BC00170=183095,975695,1075175
BC00171=183095,975695,1075175
BC00172=183095,975695,1075175
BC00173=183095,975695,1075175
BC00174=183095,975695,1075175
BC00175=183095,975695,1075175
BC00176=183095,975695,1075175
BC00177=183095,975695,1075175
BC00178=183095,975695,1075175
BC00179=210625,968928,1075175
BC00180=210625,968928,1075175
BC00181=210625,968928,1075175
BC00182=210625,968928,1075175
BC00183=210625,968928,1075175
BC00184=210625,968928,1075175
BC00185=210625,968928,1075175
BC00186=180246,951709,1075175
BC00187=180247,951710,1075174
BC00188=180247,951710,1075174
BC00189=180247,951710,1075174
BC00190=180247,951710,1075174
BC00191=180247,951710,1075174
BC00192=180247,951710,1075174
BC00193=180247,951710,1075174
BC00194=180247,951710,1075174
BC00195=180247,951710,1075174
BC00196=220770,956468,1075173
BC00197=254413,953027,1075175
BC00198=252547,954523,1075175
BC00199=252548,954519,1075175
BC00200=252583,954651,1075175
BC00201=252019,957675,1075175
BC00202=252583,954651,1075175
BC00203=252165,954787,1075175
BC00204=249030,954243,1075175
BC00205=252165,954787,1075175
BC00206=258696,949550,1075175
BC00207=257059,950024,1075175
BC00208=265795,953000,1075175
BC00209=262609,959912,1075175
BC00210=262609,959912,1075175
BC00211=262609,959912,1075175
BC00212=262609,959912,1075175
BC00213=262609,959912,1075175
BC00214=219729,982607,1075175
BC00215=219729,982607,1075175
BC00216=219729,982607,1075175
BC00217=219729,982607,1075175
BC00218=219729,982607,1075175
BC00219=219729,982607,1075175
BC00220=219729,982607,1075175
BC00221=219729,982607,1075175
BC00222=219729,982607,1075175
BC00223=219729,982607,1075175
BC00224=247259,975840,1075175
BC00225=247259,975840,1075175
BC00226=247259,975840,1075175
BC00227=247259,975840,1075175
BC00228=247259,975840,1075175
BC00229=247259,975840,1075175
BC00230=247259,975840,1075175
BC00231=216880,958621,1075175
BC00232=216881,958622,1075174
BC00233=216881,958622,1075174
BC00234=216881,958622,1075174
BC00235=216881,958622,1075174
BC00236=216881,958622,1075174
BC00237=216881,958622,1075174
BC00238=216881,958622,1075174
BC00239=216881,958622,1075174
BC00240=216881,958622,1075174
BC00241=254634,951648,1075175
BC00242=254634,951649,1075174
BC00243=254634,951649,1075174
BC00244=207516,961105,1075174
BC00245=207516,961105,1075174
BC00246=207516,961105,1075174
BC00247=207516,961105,1075174
BC00248=207516,961105,1075174
BC00249=207516,961105,1075174
BC00250=207516,961105,1075174
BC00251=207516,961105,1075174
BC00252=207675,961073,1075174
BC00253=248439,993035,1075175
BC00254=271638,1017285,1075175
BC00255=314947,1062557,1075175
BC00256=311280,1056373,1075175
BC00257=310409,1054905,1075175
BC00258=310409,1054901,1075175
BC00259=310409,1054905,1075175
BC00260=284329,1066137,1075175
BC00261=285931,1063482,1075175
BC00262=284329,1066137,1075175
BC00263=333588,1039325,1075175
BC00264=330835,1037779,1075175
BC00265=333588,1039325,1075175
BC00266=340460,1045393,1075175
BC00267=319968,1046454,1075175
BC00268=297161,1046455,1075174
BC00269=305514,1060044,1075174
BC00270=305514,1060044,1075174
BC00271=305514,1060044,1075174
BC00272=305514,1060044,1075174
BC00273=270133,1060044,1075174
BC00274=270133,1060044,1075174
BC00275=270133,1060044,1075174
BC00276=270133,1060044,1075174
BC00277=270133,1060044,1075174
BC00278=271678,1058058,1075174
BC00279=253507,1028204,1074244
BC00280=253507,1028204,1074244
BC00281=253507,1028204,1074244
BC00282=253507,1028204,1074244
BC00283=253507,1028204,1074244
BC00284=253507,1028204,1074244
BC00285=253507,1028204,1074244
BC00286=253507,1028204,1074244
BC00287=253507,1028204,1074244
BC00288=253507,1028204,1074244
BC00289=253507,1028204,1074244
BC00290=253507,1028204,1074244
BC00291=253507,1028204,1074244
BC00292=212842,1022781,1075175
BC00293=146334,1015862,1075175
BC00294=66205,1045023,1075175
BC00295=66205,1045023,1075175
BC00296=66205,1045023,1075175
BC00297=66205,1045023,1075175
BC00298=66205,1045023,1075175
BC00299=66205,1045023,1075175
BC00300=66205,1045023,1075175
BC00301=66205,1045023,1075175
BC00302=66205,1045023,1075175
BC00303=66205,1045023,1075175
BC00304=66205,1045023,1075175
BC00305=66205,1045023,1075175
BC00306=125029,959783,1075175
BC00307=190390,972133,1075175
BC00308=190390,972133,1075175
BC00309=190390,972133,1075173
BC00310=190390,972133,1075175
BC00311=190390,972133,1075175
BC00312=190390,972133,1075175
BC00313=190390,972133,1075175
BC00314=190390,972133,1075175
BC00315=190390,972133,1075175
BC00316=190390,972133,1075175
BC00317=190390,972133,1075175
BC00318=190390,972133,1075175
BC00319=190390,972133,1075175
BC00320=163122,952799,1075175
BC00321=172813,952714,1075175
BC00322=172813,952714,1075175
BC00323=172813,952714,1075175
BC00324=172813,952714,1075175
BC00325=172813,952714,1075175
BC00326=172813,952714,1075175
BC00327=172813,952714,1075175
BC00328=172813,952714,1075175
BC00329=172813,952714,1075175
BC00330=172813,952714,1075175
BC00331=172813,952714,1075175
BC00332=172813,952714,1075175
BC00333=172813,952714,1075175
BC00334=167655,947910,1075175
BC00335=103363,888035,1075175
BC00336=35304,822265,1075175
BC00337=60536,839097,1075175
BC00338=60536,839097,1075175
BC00339=60536,839097,1075175
BC00340=60536,839097,1075175
BC00341=60536,839097,1075175
BC00342=60536,839097,1075175
BC00343=35912,824089,1075175
BC00344=35912,824089,1075175
BC00345=35912,824089,1075175
BC00346=35912,824089,1075175
BC00347=35912,824089,1075175
BC00348=35912,824089,1075175
BC00349=35304,822265,1075175
BC00350=35304,822265,1075175
BC00351=35304,822265,1075175
BC00352=35304,822265,1075175
BC00353=35304,822265,1075175
BC00354=35304,822265,1075175
BC00355=35304,822265,1075175
BC00356=35304,822265,1075175
BC00357=35304,822265,1075175
BC00358=35304,822265,1075175
BC00359=35304,822265,1075175
BC00360=167967,799945,1075175
BC00361=311305,898961,1075175
BC00362=311305,898961,1075175
BC00363=311305,898961,1075175
BC00364=311305,898961,1075175
BC00365=311305,898961,1075175
BC00366=311305,898961,1075175
BC00367=311305,898961,1075175
BC00368=311305,898961,1075175
BC00369=311305,898961,1075175
BC00370=311305,898961,1075175
BC00371=311305,898961,1075175
BC00372=311305,898961,1075175
BC00373=113180,824290,1075229
BC00374=113180,824290,1075229
BC00375=113180,824290,1075229
BC00376=113180,824290,1075229
BC00377=113180,824290,1075229
BC00378=113180,824290,1075229
BC00379=113180,824290,1075229
BC00380=113180,824290,1075229
BC00381=113180,824290,1075229
BC00382=113180,824290,1075229
BC00383=113180,824290,1075229
BC00384=113180,824290,1075229
BC00385=355762,967535,1075175
BC00386=355762,967535,1075175
BC00387=355762,967535,1075175
BC00388=355762,967535,1075175
BC00389=355762,967535,1075175
BC00390=355762,967535,1075175
BC00391=355762,967535,1075175
BC00392=355762,967535,1075175
BC00393=397203,974799,1075175
BC00394=397203,974799,1075175
BC00395=397203,974799,1075175
BC00396=397203,974799,1075175
BC00397=397203,974799,1075175
BC00398=397203,974799,1075175
BC00399=397203,974799,1075175
BC00400=397203,974799,1075175
BC00401=389868,1004990,1075175
BC00402=389868,1004990,1075175
BC00403=389868,1004990,1075175
BC00404=389868,1004990,1075175
BC00405=389868,1004990,1075175
BC00406=389868,1004990,1075175
BC00407=397203,974799,1075175
BC00408=279782,952911,1075175
BC00409=264332,967435,1075175
BC00410=264332,967435,1075175
BC00411=264332,967435,1075175
BC00412=264332,967435,1075175
BC00413=264332,967435,1075175
BC00414=264332,967435,1075175
BC00415=264332,967435,1075175
BC00416=264332,967435,1075175
BC00417=264332,967435,1075175
BC00418=264332,967435,1075175
BC00419=264332,967435,1075175
BC00420=290594,956201,1075175
BC00421=316856,944967,1075175
BC00422=316856,944967,1075175
BC00423=316856,944967,1075175
BC00424=316856,944967,1075175
BC00425=316856,944967,1075175
BC00426=316856,944967,1075175
BC00427=316856,944967,1075175
BC00428=316856,944967,1075175
BC00429=316856,944967,1075175
BC00430=316856,944967,1075175
BC00431=316856,944967,1075175
BC00432=316856,944967,1075175
BC00433=316856,944967,1075175
BC00434=316856,944967,1075175
BC00435=316856,944967,1075175
BC00436=316856,944967,1075175
BC00437=329946,891084,1075175
BC00438=337525,859888,1075175
BC00439=337525,859888,1075175
BC00440=337525,859888,1075175
BC00441=337525,859888,1075175
BC00442=337525,859888,1075175
BC00443=337525,859888,1075175
BC00444=337525,859888,1075175
BC00445=337525,859888,1075175
BC00446=238148,874377,1075175
BC00447=227206,875826,1075175
BC00448=227206,875826,1075175
BC00449=227206,875826,1075175
BC00450=227206,875826,1075175
BC00451=227206,875826,1075175
BC00452=227206,875826,1075175
BC00453=280946,887675,1075175
BC00454=280946,887675,1075175
BC00455=280946,887675,1075175
BC00456=280946,887675,1075175
BC00457=280946,887675,1075175
BC00458=280946,887675,1075175
BC00459=280946,887675,1075175
BC00460=280946,887675,1075175
BC00461=239261,850045,1075175
BC00462=207869,857354,1075175
BC00463=207869,857354,1075175
BC00464=207869,857354,1075175
BC00465=207869,857354,1075175
BC00466=207869,857354,1075175
BC00467=207869,857354,1075175
BC00468=207869,857354,1075175
BC00469=207869,857354,1075175
BC00470=207996,857850,1075175
BC00471=184532,936508,1075175
BC00472=203495,1021788,1075175
BC00473=203934,1024782,1075175
BC00474=204108,1022909,1075171
BC00475=204109,1022908,1075172
BC00476=193998,1019034,1075175
BC00477=193559,1023720,1075175
BC00478=122539,997675,1075175
BC00479=122539,997675,1075175
BC00480=122540,997675,1075169
BC00481=122540,997675,1075169
BC00482=122539,997675,1075175
BC00483=122539,997675,1075175
BC00484=110261,971952,1075175
BC00485=110261,971952,1075175
BC00486=110261,971952,1075175
BC00487=110261,971952,1075175
BC00488=110261,971952,1075175
BC00489=110261,971952,1075175
BC00490=222038,980891,1075175
BC00491=314817,1023461,1075175
BC00492=333143,1031869,1075175
BC00493=333143,1031869,1075175
BC00494=333143,1031869,1075175
BC00495=333143,1031869,1075175
BC00496=333143,1031869,1075175
BC00497=163675,1006427,1075175
BC00498=163675,1006427,1075175
BC00499=164114,1001741,1075175
BC00500=164289,999867,1075175
BC00501=160191,997498,1075175
BC00502=158450,996490,1075175
BC00503=154353,994119,1075175
BC00504=154178,995993,1075175
BC00505=153739,1000679,1075175
BC00506=82719,974634,1075175
BC00507=82719,974634,1075175
BC00508=82720,974634,1075172
BC00509=82720,974634,1075172
BC00510=82719,974634,1075175
BC00511=82720,974634,1075173
BC00512=82719,974634,1075175
BC00513=82719,974634,1075175
BC00514=70441,948911,1075175
BC00515=70441,948911,1075175
BC00516=70441,948911,1075175
BC00517=70441,948911,1075175
BC00518=70441,948911,1075175
BC00519=70441,948911,1075175
BC00520=182218,957850,1075175
BC00521=274997,1000420,1075175
BC00522=293323,1008828,1075175
BC00523=293323,1008828,1075175
BC00524=293323,1008828,1075175
BC00525=293323,1008828,1075175
BC00526=293323,1008828,1075175
BC00527=293323,1008828,1075175
BC00528=337244,1059629,1075175
BC00529=337244,1059629,1075175
BC00530=337244,1059629,1075175
BC00531=337244,1059629,1075175
BC00532=337244,1059629,1075175
BC00533=337244,1059629,1075175
BC00534=337244,1059629,1075175
BC00535=227430,982125,1075175
BC00536=115014,939685,1075175
BC00537=118867,937244,1075175
BC00538=120408,936268,1075175
BC00539=124434,938528,1075175
BC00540=125926,939366,1075175
BC00541=125926,939366,1075175
BC00542=140995,947826,1075175
BC00543=140995,947826,1075175
BC00544=182041,976368,1075174
BC00545=182041,976368,1075174
BC00546=180846,977671,1075175
BC00547=177859,980929,1075175
BC00548=194800,984537,1075175
BC00549=244653,1016084,1075175
BC00550=241511,1010564,1075175
BC00551=240254,1008357,1075175
BC00552=240254,1008354,1075175
BC00553=241511,1010562,1075175
BC00554=244653,1016081,1075175
BC00555=244653,1016084,1075175
BC00556=272695,1033702,1075175
BC00557=285514,1041756,1075175
BC00558=284751,1045931,1075175
BC00559=282162,1039999,1075175
BC00560=281126,1037626,1075175
BC00561=207140,1028015,1075175
BC00562=213441,1031536,1075175
BC00563=213388,1030834,1075175
BC00564=213388,1030834,1075175
BC00565=212628,1031081,1075217
BC00566=212628,1031081,1075217
BC00567=212628,1031081,1075217
BC00568=212628,1031081,1075217
BC00569=212628,1031081,1075202
BC00570=202210,1012854,1075175
BC00571=202210,1012854,1075175
BC00572=208776,1017549,1075175
BC00573=200305,979606,1075175
BC00574=185662,909371,1075175
BC00575=185662,823633,1075175
BC00576=152631,778532,1075175
BC00577=146092,780306,1075175
BC00578=143477,781016,1075175
BC00579=143597,781078,1075175
BC00580=143625,781092,1075175
BC00581=143746,781156,1075175
BC00582=146361,780446,1075175
BC00583=152900,778672,1075175
BC00584=152900,778672,1075175
BC00585=74084,744686,1075175
BC00586=74084,744686,1075175
BC00587=67287,679894,1075175
BC00588=67287,679894,1075175
BC00589=67287,679894,1075175
BC00590=67287,679894,1075175
BC00591=67287,679894,1075175
BC00592=67287,679894,1075175
BC00593=67287,679894,1075175
BC00594=67287,679894,1075175
BC00595=83395,694294,1075175
BC00596=102108,711022,1075175
BC00597=165558,767742,1075175
BC00598=222482,818628,1075175
BC00599=215814,820321,1075175
BC00600=213147,820999,1075175
BC00601=213147,820994,1075175
BC00602=213147,820993,1075175
BC00603=213148,820988,1075175
BC00604=215815,820311,1075175
BC00605=222483,818617,1075175
BC00606=173722,816110,1075175
BC00607=90356,811823,1075175
BC00608=89696,811574,1075175
BC00609=89432,811475,1075175
BC00610=89432,811475,1075175
BC00611=89432,811475,1075175
BC00612=85301,809160,1075175
BC00613=73323,802435,1075175
BC00614=69196,800114,1075175
BC00615=69460,800213,1075175
BC00616=70120,800462,1075175
BC00617=203969,867991,1075175
BC00618=200192,866637,1075175
BC00619=198681,866095,1075175
BC00620=196278,870078,1075175
BC00621=188025,883752,1075175
BC00622=185620,887734,1075175
BC00623=187131,888276,1075175
BC00624=190907,889630,1075175
BC00625=185807,834457,1075175
BC00626=185042,826181,1075175
BC00627=182820,831186,1075175
BC00628=181931,833188,1075174
BC00629=181931,833188,1075174
BC00630=205283,846231,1075175
BC00631=205283,846231,1075175
BC00632=246906,863634,1075175
BC00633=246906,863634,1075175
BC00634=248214,861732,1075175
BC00635=251484,856977,1075175
BC00636=177002,833071,1075175
BC00637=153563,828435,1075175
BC00638=140020,825224,1075175
BC00639=143607,831260,1075175
BC00640=145042,833675,1075175
BC00641=145042,833675,1075175
BC00642=143607,831255,1075175
BC00643=140021,825218,1075175
BC00644=140020,825224,1075175
BC00645=325300,955877,1075175
BC00646=326098,960603,1075175
BC00647=326417,962494,1075175
BC00648=373942,970744,1075175
BC00649=373934,970699,1075175
BC00650=373927,970659,1075175
BC00651=372825,964128,1075175
BC00652=388713,844195,1075175
BC00653=388713,844195,1075175
BC00654=388713,844195,1075175
BC00655=388713,844195,1075175
BC00656=388713,844195,1075175
BC00657=392621,845560,1075175
BC00658=388844,869736,1075175
BC00659=388844,869736,1075175
BC00660=388844,869736,1075175
BC00661=388844,869736,1075175
BC00662=386515,859937,1075175
BC00663=382579,861240,1075175
BC00664=382579,861240,1075175
BC00665=398174,862085,1075175
BC00666=398174,860729,1075175
BC00667=398175,860364,1075172
BC00668=398174,860364,1075175
BC00669=398174,860364,1075175
BC00670=398174,860364,1075175
BC00671=398174,859798,1075175
BC00672=398174,853900,1075175
BC00673=335556,962122,1075175
BC00674=313093,960913,1075175
BC00675=312779,966350,1075175
BC00676=312653,968525,1075175
BC00677=312653,968525,1075175
BC00678=313384,968652,1075175
BC00679=313384,968652,1075175
BC00680=322722,968076,1075175
BC00681=323035,962639,1075175
BC00682=275790,965253,1075175
BC00683=219096,968390,1075175
BC00684=223120,970377,1075175
BC00685=224729,971172,1075175
BC00686=224729,971172,1075175
BC00687=224591,971007,1075175
BC00688=224591,971007,1075175
BC00689=219210,965708,1075175
BC00690=215186,963721,1075175
BC00691=283252,975030,1075175
BC00692=343583,985054,1075175
BC00693=351318,986339,1075175
BC00694=346951,987672,1075175
BC00695=346840,986833,1075175
BC00696=346840,986833,1075175
BC00697=346840,986832,1075174
BC00698=346840,986832,1075174
BC00699=346840,986832,1075174
BC00700=351469,983882,1075175
BC00701=355836,982549,1075175
BC00702=351318,986339,1075175
BC00703=375376,962122,1075175
BC00704=352913,960913,1075175
BC00705=352599,966350,1075175
BC00706=352473,968525,1075175
BC00707=352473,968525,1075175
BC00708=352749,968573,1075175
BC00709=352749,968573,1075175
BC00710=362542,968076,1075175
BC00711=362855,962639,1075175
BC00712=315610,965253,1075175
BC00713=258916,968390,1075175
BC00714=262940,970377,1075175
BC00715=264549,993234,1075175
BC00716=264533,993126,1075175
BC00717=264533,993126,1075175
BC00718=264533,993126,1075175
BC00719=259030,965708,1075175
BC00720=255006,963721,1075175
BC00721=323072,975030,1075175
BC00722=383403,985054,1075175
BC00723=391138,986339,1075175
BC00724=386771,987672,1075175
BC00725=385397,987893,1075175
BC00726=385397,987893,1075175
BC00727=385397,987893,1075175
BC00728=385397,987893,1075175
BC00729=391289,983882,1075175
BC00730=394785,983280,1075175
BC00731=393350,984484,1075175
BC00732=322594,894090,1075175
BC00733=319270,885244,1075175
BC00734=319145,881395,1075175
BC00735=319096,879856,1075175
BC00736=319096,879856,1075175
BC00737=310158,881364,1075175
BC00738=310282,885213,1075175
BC00739=287932,898047,1075175
BC00740=289217,893542,1075175
BC00741=289730,891739,1075175
BC00742=285692,891718,1075175
BC00743=285179,893520,1075175
BC00744=283894,898026,1075175
BC00745=317886,904348,1075175
BC00746=321408,904356,1075175
BC00747=251917,914686,1075175
BC00748=191223,885215,1075175
BC00749=191223,923708,1075175
BC00750=186619,926680,1075175
BC00751=184777,927869,1075175
BC00752=132357,904545,1075175
BC00753=148459,907340,1075175
BC00754=150318,907039,1075175
BC00755=172119,903510,1075175
BC00756=172334,901853,1075175
BC00757=172871,897709,1075175
BC00758=285135,920733,1075175
BC00759=282294,924718,1075175
BC00760=278369,925274,1075175
BC00761=250842,915028,1075175
BC00762=259644,916574,1075175
BC00763=259644,916574,1075174
BC00764=259644,916574,1075175
BC00765=285135,920733,1075175
BC00766=320470,920733,1075175
BC00767=320470,920733,1075175
BC00768=320470,920733,1075172
BC00769=320470,920733,1075172
BC00770=320470,920733,1075172
BC00771=302481,924098,1075175
BC00772=235391,926007,1075175
BC00773=235391,926007,1075175
BC00774=227742,920504,1075175
BC00775=172871,874776,1075175
BC00776=140749,823212,1075175
BC00777=114392,780903,1075175
BC00778=114392,780903,1075175
BC00779=114392,780903,1075175
BC00780=114392,780903,1075175
BC00781=114393,780903,1075175
BC00782=114392,780903,1075175
BC00783=114392,780903,1075175
BC00784=114392,780903,1075175
BC00785=147421,791636,1075175
BC00786=157474,794903,1075175
BC00787=157474,794903,1075175
BC00788=157474,794903,1075174
BC00789=157474,794903,1075175
BC00790=157474,794903,1075175
BC00791=157474,794903,1075175
BC00792=157474,794903,1075175
BC00793=157474,794903,1075175
BC00794=188976,808930,1075175
BC00795=188976,808930,1075175
BC00796=188976,808930,1075175
BC00797=188976,808930,1075175
BC00798=188976,808930,1075175
BC00799=188976,808930,1075175
BC00800=188976,808930,1075175
BC00801=188976,808930,1075175
BC00802=147641,782026,1075175
BC00803=198576,845167,1075175
BC00804=232811,933878,1075175
BC00805=232896,933343,1075175
BC00806=232035,938717,1075175
BC00807=231691,940867,1075175
BC00808=233684,941999,1075172
BC00809=218918,951560,1075175
BC00810=218487,945823,1075175
BC00811=199715,965567,1075175
BC00812=202231,971242,1075175
BC00813=203237,973512,1075175
BC00814=199770,971953,1075175
BC00815=198686,969649,1075175
BC00816=195975,963887,1075175
BC00817=268319,958805,1075175
BC00818=299772,956595,1075175
BC00819=294961,960779,1075175
BC00820=302025,967105,1075175
BC00821=302025,967105,1075175
BC00822=302862,967571,1075175
BC00823=304981,965989,1075175
BC00824=310277,962032,1075175
BC00825=299772,946803,1075175
BC00826=156368,867370,1075175
BC00827=114190,943890,1075175
BC00828=112857,947238,1075175
BC00829=112324,948578,1075175
BC00830=112324,948578,1075175
BC00831=97258,945962,1075175
BC00832=58795,939285,1075175
BC00833=58795,939285,1075175
BC00834=57972,937710,1075175
BC00835=59304,934362,1075175
BC00836=59959,931573,1075175
BC00837=60163,930702,1075175
BC00838=64900,934429,1075175
BC00839=66794,935919,1075175
BC00840=70926,933782,1075175
BC00841=86714,920781,1075175
BC00842=88876,916896,1075175
BC00843=87247,915034,1075175
BC00844=83174,910378,1075175
BC00845=93083,910762,1075175
BC00846=96362,916987,1075175
BC00847=99439,917931,1075175
BC00848=102107,915596,1075175
BC00849=93734,925368,1075175
BC00850=92128,923198,1075175
BC00851=88115,917772,1075175
BC00852=59304,853852,1075175
BC00853=302197,956351,1075175
BC00854=302197,956351,1075175
BC00855=297684,958955,1075175
BC00856=295879,959997,1075175
BC00857=304739,998959,1075175
BC00858=304739,998896,1075175
BC00859=293949,1042099,1075175
BC00860=295296,1044279,1075175
BC00861=298665,1049727,1075175
BC00862=298665,1049727,1075175
BC00863=302197,956351,1075175
BC00864=339931,956351,1075175
BC00865=339931,956351,1075175
BC00866=339931,956351,1075175
BC00867=345108,996833,1075175
BC00868=329498,1037164,1075167
BC00869=329498,1037164,1075167
BC00870=329498,1037164,1075167
BC00871=326051,1024211,1075168
BC00872=315665,949153,1075168
BC00873=252444,896504,1075168
BC00874=116643,896504,1075168
BC00875=116643,972299,1075168
BC00876=116644,972299,1070754
BC00877=116644,972299,1070754
BC00878=121804,1001122,1070754
BC00879=121804,1001122,1070754
BC00880=121804,1001122,1070754
BC00881=121804,1001122,1070754
BC00882=164206,909682,1070754
BC00883=118737,834368,1072160
BC00884=21214,672831,1075175
BC00885=78393,670967,1075175
BC00886=177059,727519,1002542
BC00887=78393,913126,1075175
BC00888=70793,903989,1075175
BC00889=70793,903989,1075175
BC00890=70793,903989,1075175
BC00891=70793,903989,1075175
BC00892=70793,903989,1075175
BC00893=70793,903989,1075175
BC00894=70793,903989,1075175
BC00895=70793,903989,1075175
BC00896=70793,903989,1075175
BC00897=103901,897249,1075175
BC00898=103901,897249,1075175
BC00899=103901,897249,1075175
BC00900=103901,897249,1075175
BC00901=103901,897249,1075175
BC00902=103901,897249,1075175
BC00903=103901,897249,1075175
BC00904=103901,897249,1075175
BC00905=89915,910531,1075175
BC00906=89915,910531,1075175
BC00907=89915,910531,1075175
BC00908=89915,910531,1075175
BC00909=89915,910531,1075175
BC00910=89915,910531,1075175
BC00911=89915,910531,1075175
BC00912=89915,910531,1075175
BC00913=89915,910531,1075175
BC00914=27368,899646,1075175
BC00915=27368,899646,1075175
BC00916=27368,899646,1075175
BC00917=27368,899646,1075175
BC00918=27368,899646,1075175
BC00919=27368,899646,1075175
BC00920=27368,899646,1075175
BC00921=27368,899646,1075175
BC00922=160753,772187,1075175
BC00923=160753,772187,1075175
BC00924=160753,772187,1075175
BC00925=160753,772187,1075175
BC00926=160753,772187,1075175
BC00927=160753,772187,1075175
BC00928=160753,772187,1075175
BC00929=160753,772187,1075175
BC00930=160753,772187,1075175
BC00931=160753,772187,1075175
BC00932=160753,772187,1075175
BC00933=160753,772187,1075175
BC00934=123402,765716,1075175
BC00935=123402,765716,1075175
BC00936=123402,765716,1075175
BC00937=123402,765716,1075175
BC00938=123402,765716,1075175
BC00939=123402,765716,1075175
BC00940=123402,765716,1075175
BC00941=123402,765716,1075175
BC00942=123402,765716,1075175
BC00943=123402,765716,1075175
BC00944=123402,765716,1075175
BC00945=129464,768278,1075175
BC00946=151149,777443,1075175
BC00947=169689,785624,1075175
BC00948=169689,785624,1075175
BC00949=169689,785624,1075175
BC00950=169689,785624,1075175
BC00951=169689,785624,1075175
BC00952=169689,785624,1075175
BC00953=169689,785624,1075175
BC00954=169689,785624,1075175
BC00955=169689,785624,1075175
BC00956=169689,785624,1075175
BC00957=169689,785624,1075175
BC00958=169689,785624,1075175
BC00959=169689,785624,1075175
BC00960=120114,813651,1075175
BC00961=120114,813651,1075175
BC00962=120114,813651,1075175
BC00963=120114,813651,1075175
BC00964=120114,813651,1075175
BC00965=120114,813651,1075175
BC00966=120114,813651,1075175
BC00967=120114,813651,1075175
BC00968=120114,813651,1075175
BC00969=120114,813651,1075175
BC00970=120114,813651,1075175
BC00971=120114,813651,1075175
BC00972=120114,813651,1075175
BC00973=141881,838168,1075175
BC00974=141881,838168,1075175
BC00975=141881,838168,1075175
BC00976=141881,838168,1075175
BC00977=141881,838168,1075175
BC00978=141881,838168,1075175
BC00979=141881,838168,1075175
BC00980=141881,838168,1075175
BC00981=141881,838168,1075175
BC00982=141881,838168,1075175
BC00983=141881,838168,1075175
BC00984=141881,838168,1075175
BC00985=141881,838168,1075175
BC00986=69874,805894,1075175
BC00987=70019,750208,1075175
BC00988=70019,750208,1075175
BC00989=70019,750208,1075175
BC00990=70019,750208,1075175
BC00991=70019,750208,1075175
BC00992=70019,750208,1075175
BC00993=70019,750208,1075175
BC00994=70019,750208,1075175
BC00995=70019,750208,1075175
BC00996=70019,750208,1075175
BC00997=70019,750208,1075175
BC00998=70019,750208,1075175
BC00999=70019,750208,1075175
BC01000=70018,750208,1075172
BC01001=70018,750208,1075172
BC01002=70018,750208,1075172
BC01003=70018,750208,1075172
BC01004=70018,750208,1075172
BC01005=70018,750208,1075172
BC01006=70018,750208,1075172
BC01007=70018,750208,1075172
BC01008=110204,822960,1075174
BC01009=128430,855958,1075175
BC01010=125005,945340,1075175
BC01011=125005,945340,1075175
BC01012=125005,945340,1075175
BC01013=125005,945340,1075175
BC01014=125005,945340,1075175
BC01015=125005,945340,1075175
BC01016=125005,945340,1075175
BC01017=125005,945340,1075175
BC01018=125005,945340,1075175
BC01019=125005,945340,1075175
BC01020=125005,945340,1075175
BC01021=177748,940008,1075175
BC01022=177748,940008,1075175
BC01023=177748,940008,1075175
BC01024=177748,940008,1075175
BC01025=177748,940008,1075175
BC01026=177748,940008,1075175
BC01027=177748,940008,1075175
BC01028=177748,940008,1075175
BC01029=177748,940008,1075175
BC01030=177748,940008,1075175
BC01031=177748,940008,1075175
BC01032=177748,940008,1075175
BC01033=225975,953000,1075175
BC01034=225975,953000,1075175
BC01035=225975,953000,1075175
BC01036=225975,953000,1075175
BC01037=225975,953000,1075175
BC01038=225975,953000,1075175
BC01039=225975,953000,1075175
BC01040=225975,953000,1075175
BC01041=225975,953000,1075175
BC01042=225975,953000,1075175
BC01043=225975,953000,1075175
BC01044=225975,953000,1075175
BC01045=254413,953027,1075175
BC01046=252547,954523,1075175
BC01047=252548,954519,1075175
BC01048=252583,954651,1075175
BC01049=252019,957675,1075175
BC01050=252583,954651,1075175
BC01051=252165,954787,1075175
BC01052=249030,954243,1075175
BC01053=252165,954787,1075175
BC01054=258696,949550,1075175
BC01055=257059,950024,1075175
BC01056=265795,953000,1075175
BC01057=265795,953000,1075175
BC01058=265795,953000,1075175
BC01059=265795,953000,1075175
BC01060=265795,953000,1075175
BC01061=265795,953000,1075175
BC01062=265795,953000,1075175
BC01063=265795,953000,1075175
BC01064=265795,953000,1075175
BC01065=265795,953000,1075175
BC01066=265795,953000,1075175
BC01067=254634,951648,1075175
BC01068=253737,956448,1075175
BC01069=253378,958368,1075175
BC01070=253379,958364,1075175
BC01071=253259,958395,1075175
BC01072=252695,961419,1075175
BC01073=253259,958395,1075175
BC01074=254515,951675,1075175
BC01075=248439,993035,1075175
BC01076=271638,1017285,1075175
BC01077=314947,1062557,1075175
BC01078=311280,1056373,1075175
BC01079=310409,1054905,1075175
BC01080=310409,1054901,1075175
BC01081=310409,1054905,1075175
BC01082=284329,1066137,1075175
BC01083=285931,1063482,1075175
BC01084=284329,1066137,1075175
BC01085=333588,1039325,1075175
BC01086=330835,1037779,1075175
BC01087=333588,1039325,1075175
BC01088=340460,1045393,1075175
BC01089=319968,1046454,1075175
BC01090=279319,1048558,1075175
BC01091=281895,1044284,1075175
BC01092=282926,1042574,1075175
BC01093=282926,1042570,1075175
BC01094=282744,1042486,1075175
BC01095=284346,1039831,1075175
BC01096=282744,1042486,1075175
BC01097=279137,1048470,1075175
BC01098=253507,1028204,1074244
BC01099=253507,1028204,1074244
BC01100=253507,1028204,1074244
BC01101=253507,1028204,1074244
BC01102=253507,1028204,1074244
BC01103=253507,1028204,1074244
BC01104=253507,1028204,1074244
BC01105=253507,1028204,1074244
BC01106=253507,1028204,1074244
BC01107=253507,1028204,1074244
BC01108=253507,1028204,1074244
BC01109=253507,1028204,1074244
BC01110=253507,1028204,1074244
BC01111=212842,1022781,1075175
BC01112=146334,1015862,1075175
BC01113=66205,1045023,1075175
BC01114=66205,1045023,1075175
BC01115=66205,1045023,1075175
BC01116=66205,1045023,1075175
BC01117=66205,1045023,1075175
BC01118=66205,1045023,1075175
BC01119=66205,1045023,1075175
BC01120=66205,1045023,1075175
BC01121=66205,1045023,1075175
BC01122=66205,1045023,1075175
BC01123=66205,1045023,1075175
BC01124=66205,1045023,1075175
BC01125=125029,959783,1075175
BC01126=190390,972133,1075175
BC01127=190390,972133,1075175
BC01128=190390,972133,1075173
BC01129=190390,972133,1075175
BC01130=190390,972133,1075175
BC01131=190390,972133,1075175
BC01132=190390,972133,1075175
BC01133=190390,972133,1075175
BC01134=190390,972133,1075175
BC01135=190390,972133,1075175
BC01136=190390,972133,1075175
BC01137=190390,972133,1075175
BC01138=190390,972133,1075175
BC01139=103363,888035,1075175
BC01140=35304,822265,1075175
BC01141=35304,822265,1075175
BC01142=35304,822265,1075175
BC01143=35304,822265,1075175
BC01144=35304,822265,1075175
BC01145=35304,822265,1075175
BC01146=35304,822265,1075175
BC01147=35304,822265,1075175
BC01148=35304,822265,1075175
BC01149=35304,822265,1075175
BC01150=35304,822265,1075175
BC01151=35304,822265,1075175
BC01152=167967,799945,1075175
BC01153=311305,898961,1075175
BC01154=311305,898961,1075175
BC01155=311305,898961,1075175
BC01156=311305,898961,1075175
BC01157=311305,898961,1075175
BC01158=311305,898961,1075175
BC01159=311305,898961,1075175
BC01160=311305,898961,1075175
BC01161=311305,898961,1075175
BC01162=311305,898961,1075175
BC01163=311305,898961,1075175
BC01164=311305,898961,1075175
BC01165=113180,824290,1075229
BC01166=113180,824290,1075229
BC01167=113180,824290,1075229
BC01168=113180,824290,1075229
BC01169=113180,824290,1075229
BC01170=113180,824290,1075229
BC01171=113180,824290,1075229
BC01172=113180,824290,1075229
BC01173=113180,824290,1075229
BC01174=113180,824290,1075229
BC01175=113180,824290,1075229
BC01176=113180,824290,1075229
BC01177=355762,967535,1075175
BC01178=355762,967535,1075175
BC01179=355762,967535,1075175
BC01180=355762,967535,1075175
BC01181=355762,967535,1075175
BC01182=355762,967535,1075175
BC01183=355762,967535,1075175
BC01184=355762,967535,1075175
BC01185=397203,974799,1075175
BC01186=397203,974799,1075175
BC01187=397203,974799,1075175
BC01188=397203,974799,1075175
BC01189=397203,974799,1075175
BC01190=397203,974799,1075175
BC01191=397203,974799,1075175
BC01192=397203,974799,1075175
BC01193=279782,952911,1075175
BC01194=264332,967435,1075175
BC01195=264332,967435,1075175
BC01196=264332,967435,1075175
BC01197=264332,967435,1075175
BC01198=264332,967435,1075175
BC01199=264332,967435,1075175
BC01200=264332,967435,1075175
BC01201=264332,967435,1075175
BC01202=264332,967435,1075175
BC01203=264332,967435,1075175
BC01204=264332,967435,1075175
BC01205=290594,956201,1075175
BC01206=316856,944967,1075175
BC01207=316856,944967,1075175
BC01208=316856,944967,1075175
BC01209=316856,944967,1075175
BC01210=316856,944967,1075175
BC01211=316856,944967,1075175
BC01212=316856,944967,1075175
BC01213=316856,944967,1075175
BC01214=316856,944967,1075175
BC01215=316856,944967,1075175
BC01216=316856,944967,1075175
BC01217=316856,944967,1075175
BC01218=316856,944967,1075175
BC01219=316856,944967,1075175
BC01220=316856,944967,1075175
BC01221=316856,944967,1075175
BC01222=329946,891084,1075175
BC01223=337525,859888,1075175
BC01224=337525,859888,1075175
BC01225=337525,859888,1075175
BC01226=337525,859888,1075175
BC01227=337525,859888,1075175
BC01228=337525,859888,1075175
BC01229=337525,859888,1075175
BC01230=337525,859888,1075175
BC01231=238148,874377,1075175
BC01232=227206,875826,1075175
BC01233=227206,875826,1075175
BC01234=227206,875826,1075175
BC01235=227206,875826,1075175
BC01236=227206,875826,1075175
BC01237=227206,875826,1075175
BC01238=280946,887675,1075175
BC01239=280946,887675,1075175
BC01240=280946,887675,1075175
BC01241=280946,887675,1075175
BC01242=280946,887675,1075175
BC01243=280946,887675,1075175
BC01244=280946,887675,1075175
BC01245=280946,887675,1075175
BC01246=239261,850045,1075175
BC01247=207869,857354,1075175
BC01248=207869,857354,1075175
BC01249=207869,857354,1075175
BC01250=207869,857354,1075175
BC01251=207869,857354,1075175
BC01252=207869,857354,1075175
BC01253=207869,857354,1075175
BC01254=207869,857354,1075175
BC01255=207996,857850,1075175
BC01256=184532,936508,1075175
BC01257=203495,1021788,1075175
BC01258=203934,1024782,1075175
BC01259=204108,1022909,1075171
BC01260=204109,1022908,1075172
BC01261=193998,1019034,1075175
BC01262=193559,1023720,1075175
BC01263=122539,997675,1075175
BC01264=122539,997675,1075175
BC01265=122540,997675,1075169
BC01266=122540,997675,1075169
BC01267=122539,997675,1075175
BC01268=122539,997675,1075175
BC01269=110261,971952,1075175
BC01270=110261,971952,1075175
BC01271=110261,971952,1075175
BC01272=110261,971952,1075175
BC01273=110261,971952,1075175
BC01274=110261,971952,1075175
BC01275=222038,980891,1075175
BC01276=314817,1023461,1075175
BC01277=333143,1031869,1075175
BC01278=333143,1031869,1075175
BC01279=333143,1031869,1075175
BC01280=333143,1031869,1075175
BC01281=333143,1031869,1075175
BC01282=163675,1006427,1075175
BC01283=163675,1006427,1075175
BC01284=164114,1001741,1075175
BC01285=164289,999867,1075175
BC01286=160191,997498,1075175
BC01287=158450,996490,1075175
BC01288=154353,994119,1075175
BC01289=154178,995993,1075175
BC01290=153739,1000679,1075175
BC01291=82719,974634,1075175
BC01292=82719,974634,1075175
BC01293=82720,974634,1075172
BC01294=82720,974634,1075172
BC01295=82719,974634,1075175
BC01296=82720,974634,1075173
BC01297=82719,974634,1075175
BC01298=82719,974634,1075175
BC01299=70441,948911,1075175
BC01300=70441,948911,1075175
BC01301=70441,948911,1075175
BC01302=70441,948911,1075175
BC01303=70441,948911,1075175
BC01304=70441,948911,1075175
BC01305=182218,957850,1075175
BC01306=274997,1000420,1075175
BC01307=293323,1008828,1075175
BC01308=293323,1008828,1075175
BC01309=293323,1008828,1075175
BC01310=293323,1008828,1075175
BC01311=293323,1008828,1075175
BC01312=293323,1008828,1075175
BC01313=337244,1059629,1075175
BC01314=337244,1059629,1075175
BC01315=337244,1059629,1075175
BC01316=337244,1059629,1075175
BC01317=337244,1059629,1075175
BC01318=337244,1059629,1075175
BC01319=337244,1059629,1075175
BC01320=227430,982125,1075175
BC01321=115014,939685,1075175
BC01322=118867,937244,1075175
BC01323=120408,936268,1075175
BC01324=140995,947826,1075175
BC01325=182041,976368,1075175
BC01326=180846,977671,1075175
BC01327=177859,980929,1075175
BC01328=194800,984537,1075175
BC01329=244653,1016084,1075175
BC01330=241511,1010564,1075175
BC01331=240254,1008357,1075175
BC01332=240254,1008354,1075175
BC01333=241511,1010562,1075175
BC01334=244653,1016081,1075175
BC01335=244653,1016084,1075175
BC01336=272695,1033702,1075175
BC01337=285514,1041756,1075175
BC01338=284751,1045931,1075175
BC01339=282162,1039999,1075175
BC01340=281126,1037626,1075175
BC01341=207140,1028015,1075175
BC01342=213441,1031536,1075175
BC01343=213388,1030834,1075175
BC01344=213388,1030834,1075175
BC01345=212628,1031081,1075217
BC01346=212628,1031081,1075217
BC01347=212628,1031081,1075217
BC01348=212628,1031081,1075217
BC01349=212628,1031081,1075202
BC01350=202210,1012854,1075175
BC01351=202210,1012854,1075175
BC01352=196613,982513,1075175
BC01353=175963,870568,1075175
BC01354=163612,803610,1075175
BC01355=152631,778532,1075175
BC01356=146092,780306,1075175
BC01357=143477,781016,1075175
BC01358=143597,781078,1075175
BC01359=143625,781092,1075175
BC01360=143746,781156,1075175
BC01361=146361,780446,1075175
BC01362=152900,778672,1075175
BC01363=152900,778672,1075175
BC01364=74084,744686,1075175
BC01365=74084,744686,1075175
BC01366=67287,679894,1075175
BC01367=67287,679894,1075175
BC01368=67287,679894,1075175
BC01369=67287,679894,1075175
BC01370=67287,679894,1075175
BC01371=67287,679894,1075175
BC01372=67287,679894,1075175
BC01373=67287,679894,1075175
BC01374=83395,694294,1075175
BC01375=102108,711022,1075175
BC01376=165558,767742,1075175
BC01377=222482,818628,1075175
BC01378=215814,820321,1075175
BC01379=213147,820999,1075175
BC01380=213147,820994,1075175
BC01381=213147,820993,1075175
BC01382=213148,820988,1075175
BC01383=215815,820311,1075175
BC01384=222483,818617,1075175
BC01385=173722,816110,1075175
BC01386=90356,811823,1075175
BC01387=89696,811574,1075175
BC01388=89432,811475,1075175
BC01389=85301,809160,1075175
BC01390=73323,802435,1075175
BC01391=69196,800114,1075175
BC01392=69460,800213,1075175
BC01393=70120,800462,1075175
BC01394=203969,867991,1075175
BC01395=200192,866637,1075175
BC01396=198681,866095,1075175
BC01397=196278,870078,1075175
BC01398=188025,883752,1075175
BC01399=185620,887734,1075175
BC01400=187131,888276,1075175
BC01401=190907,889630,1075175
BC01402=185807,834457,1075175
BC01403=185042,826181,1075175
BC01404=182820,831186,1075175
BC01405=181931,833188,1075175
BC01406=205283,846231,1075175
BC01407=246906,863634,1075175
BC01408=246906,863634,1075175
BC01409=248214,861732,1075175
BC01410=251484,856977,1075175
BC01411=177002,833071,1075175
BC01412=153563,828435,1075175
BC01413=140020,825224,1075175
BC01414=143607,831260,1075175
BC01415=145042,833675,1075175
BC01416=145042,833669,1075175
BC01417=143607,831255,1075175
BC01418=140021,825218,1075175
BC01419=140020,825224,1075175
BC01420=325300,955877,1075175
BC01421=326098,960603,1075175
BC01422=326417,962494,1075175
BC01423=373942,970744,1075175
BC01424=373623,968854,1075175
BC01425=372825,964128,1075175
BC01426=388713,844195,1075175
BC01427=388713,844195,1075175
BC01428=388713,844195,1075175
BC01429=388713,844195,1075175
BC01430=388713,844195,1075175
BC01431=392621,845560,1075175
BC01432=388844,869736,1075175
BC01433=388844,869736,1075175
BC01434=388844,869736,1075175
BC01435=388844,869736,1075175
BC01436=386515,859937,1075175
BC01437=382579,861240,1075175
BC01438=382579,861240,1075175
BC01439=398174,862085,1075175
BC01440=398174,860729,1075175
BC01441=398175,860364,1075172
BC01442=398174,860364,1075175
BC01443=398174,860364,1075175
BC01444=398174,860364,1075175
BC01445=398174,859798,1075175
BC01446=398174,853900,1075175
BC01447=335556,962122,1075175
BC01448=313093,960913,1075175
BC01449=312779,966350,1075175
BC01450=312653,968525,1075175
BC01451=317356,969341,1075175
BC01452=322596,970251,1075175
BC01453=322722,968076,1075175
BC01454=323035,962639,1075175
BC01455=275790,965253,1075175
BC01456=219096,968390,1075175
BC01457=223120,970377,1075175
BC01458=224729,971172,1075175
BC01459=220819,966503,1075175
BC01460=219210,965708,1075175
BC01461=215186,963721,1075175
BC01462=283252,975030,1075175
BC01463=343583,985054,1075175
BC01464=351318,986339,1075175
BC01465=346951,987672,1075175
BC01466=345577,987893,1075175
BC01467=346840,986833,1075175
BC01468=348087,985787,1075175
BC01469=349722,984415,1075175
BC01470=349722,984415,1075175
BC01471=349722,984415,1075175
BC01472=351469,983882,1075175
BC01473=355836,982549,1075175
BC01474=351318,986339,1075175
BC01475=375376,962122,1075175
BC01476=352913,960913,1075175
BC01477=352599,966350,1075175
BC01478=352473,968525,1075175
BC01479=357176,969341,1075175
BC01480=362416,970251,1075175
BC01481=362542,968076,1075175
BC01482=362855,962639,1075175
BC01483=315610,965253,1075175
BC01484=258916,968390,1075175
BC01485=262940,970377,1075175
BC01486=264549,971172,1075175
BC01487=260639,966503,1075175
BC01488=259030,965708,1075175
BC01489=255006,963721,1075175
BC01490=323072,975030,1075175
BC01491=383403,985054,1075175
BC01492=391138,986339,1075175
BC01493=386771,987672,1075175
BC01494=385397,987893,1075175
BC01495=386660,986833,1075175
BC01496=387907,985787,1075175
BC01497=389542,984415,1075175
BC01498=389542,984415,1075175
BC01499=389542,984415,1075175
BC01500=391289,983882,1075175
BC01501=394785,983280,1075175
BC01502=393350,984484,1075175
BC01503=322594,894090,1075175
BC01504=319270,885244,1075175
BC01505=319145,881395,1075175
BC01506=319096,879856,1075175
BC01507=319096,879856,1075175
BC01508=310158,881364,1075175
BC01509=310282,885213,1075175
BC01510=287932,898047,1075175
BC01511=289217,893542,1075175
BC01512=289730,891739,1075175
BC01513=285692,891718,1075175
BC01514=285179,893520,1075175
BC01515=283894,898026,1075175
BC01516=317886,904348,1075175
BC01517=321408,904356,1075175
BC01518=251917,914686,1075175
BC01519=191223,885215,1075175
BC01520=191223,923708,1075175
BC01521=186619,926680,1075175
BC01522=184777,927869,1075175
BC01523=132357,904545,1075175
BC01524=148459,907340,1075175
BC01525=150318,907039,1075175
BC01526=172119,903510,1075175
BC01527=172334,901853,1075175
BC01528=172871,897709,1075175
BC01529=285135,920733,1075175
BC01530=282294,924718,1075175
BC01531=278369,925274,1075175
BC01532=250842,915028,1075175
BC01533=259644,916574,1075175
BC01534=259644,916574,1075174
BC01535=259644,916574,1075175
BC01536=285135,920733,1075175
BC01537=320470,920733,1075175
BC01538=320470,920733,1075175
BC01539=320470,920733,1075172
BC01540=320470,920733,1075172
BC01541=320470,920733,1075172
BC01542=302481,924098,1075175
BC01543=235391,926007,1075175
BC01544=235391,926007,1075175
BC01545=227742,920504,1075175
BC01546=172871,874776,1075175
BC01547=140749,823212,1075175
BC01548=114392,780903,1075175
BC01549=114392,780903,1075175
BC01550=114392,780903,1075175
BC01551=114392,780903,1075175
BC01552=114392,780903,1075175
BC01553=114392,780903,1075175
BC01554=114392,780903,1075175
BC01555=114392,780903,1075175
BC01556=147421,791636,1075175
BC01557=157474,794903,1075175
BC01558=157474,794903,1075175
BC01559=157474,794903,1075175
BC01560=157474,794903,1075175
BC01561=157474,794903,1075175
BC01562=157474,794903,1075175
BC01563=157474,794903,1075175
BC01564=157474,794903,1075175
BC01565=188976,808930,1075175
BC01566=188976,808930,1075175
BC01567=188976,808930,1075175
BC01568=188976,808930,1075175
BC01569=188976,808930,1075175
BC01570=188976,808930,1075175
BC01571=188976,808930,1075175
BC01572=188976,808930,1075175
BC01573=147641,782026,1075175
BC01574=198576,845167,1075175
BC01575=232811,933878,1075175
BC01576=232896,933343,1075175
BC01577=232035,938717,1075175
BC01578=231691,940867,1075175
BC01579=233684,941999,1075172
BC01580=218918,951560,1075175
BC01581=218487,945823,1075175
BC01582=199715,965567,1075175
BC01583=202231,971242,1075175
BC01584=203237,973512,1075175
BC01585=199770,971953,1075175
BC01586=198686,969649,1075175
BC01587=195975,963887,1075175
BC01588=268319,958805,1075175
BC01589=299772,956595,1075175
BC01590=294961,960779,1075175
BC01591=302025,967105,1075175
BC01592=302025,967105,1075175
BC01593=302862,967571,1075175
BC01594=304981,965989,1075175
BC01595=310277,962032,1075175
BC01596=299772,946803,1075175
BC01597=156368,867370,1075175
BC01598=114190,943890,1075175
BC01599=112857,947238,1075175
BC01600=112324,948578,1075175
BC01601=57438,939049,1075175
BC01602=57438,939049,1075175
BC01603=57972,937710,1075175
BC01604=59304,934362,1075175
BC01605=59959,931573,1075175
BC01606=60163,930702,1075175
BC01607=64900,934429,1075175
BC01608=66794,935919,1075175
BC01609=70926,933782,1075175
BC01610=86714,920781,1075175
BC01611=88876,916896,1075175
BC01612=87247,915034,1075175
BC01613=83174,910378,1075175
BC01614=93083,910762,1075175
BC01615=96362,916987,1075175
BC01616=97673,919477,1075175
BC01617=102107,915596,1075175
BC01618=93734,925368,1075175
BC01619=92128,923198,1075175
BC01620=88115,917772,1075175
BC01621=59304,853852,1075175
BC01622=302197,956351,1075175
BC01623=302197,956351,1075175
BC01624=297684,958955,1075175
BC01625=295879,959997,1075175
BC01626=304739,998959,1075175
BC01627=304723,978619,1075175
BC01628=293949,1042099,1075175
BC01629=295296,1044279,1075175
BC01630=298665,1049727,1075175
BC01631=298665,1049727,1075175
BC01632=302197,956351,1075175
BC01633=339931,956351,1075175
BC01634=339931,956351,1075175
BC01635=339931,956351,1075175
BC01636=345108,996833,1075175
BC01637=329498,1037164,1075167
BC01638=329498,1037164,1075167
BC01639=329498,1037164,1075167
BC01640=326051,1024211,1075168
BC01641=315665,949153,1075168
BC01642=252444,896504,1075168
BC01643=116643,896504,1075168
BC01644=116643,972299,1075168
BC01645=116644,972299,1070754
BC01646=116644,972299,1070754
BC01647=121804,1001122,1070754
BC01648=121804,1001122,1070754
BC01649=121804,1001122,1070754
BC01650=121804,1001122,1070754
BC01651=164206,909682,1070754
BC01652=118737,834368,1072160
BC01653=21214,672831,1075175
BC01654=21214,672831,272422
BC01655=236199,677421,175874
BC01656=277013,737492,108841
BC01657=313151,790681,49489
BC01658=313151,790681,49489
BC01659=313151,790681,49489
BC01660=313151,790681,49489
BC01661=313151,790681,49489
BC01662=313151,790681,49489
BC01663=313151,790681,49489
BC01664=313151,790681,49489
BC01665=313151,790681,49489
BC01666=339082,790681,219047
BC01667=339082,790681,219047
BC01668=339082,790681,219047
BC01669=339082,790681,219047
BC01670=339082,790681,219047
BC01671=339082,790681,219047
BC01672=339082,790681,219047
BC01673=339082,790681,219047
BC01674=339082,790681,219047
BC01675=318756,790681,206942
BC01676=318756,790681,206942
BC01677=318756,790681,206942
BC01678=318756,790681,206942
BC01679=318756,790681,206942
BC01680=318756,790681,206942
BC01681=318756,790681,206941
BC01682=318756,790681,206941
BC01683=318756,790681,206942
BC01684=330178,790681,186109
BC01685=360333,790681,131110
BC01686=360333,790681,131110
BC01687=360333,790681,131110
BC01688=360333,790681,131110
BC01689=360333,790681,131110
BC01690=360333,790681,131110
BC01691=360333,790681,131110
BC01692=360333,790681,131110
BC01693=360333,790681,131110
BC01694=319787,790681,204440
BC01695=319787,790681,204440
BC01696=319787,790681,204440
BC01697=319787,790681,204440
BC01698=319787,790681,204440
BC01699=319787,790681,204440
BC01700=319787,790681,204440
BC01701=319787,790681,204440
BC01702=319787,790681,204440
BC01703=319787,790681,204440
BC01704=345989,790681,139065
BC01705=345989,790681,139065
BC01706=345989,790681,139065
BC01707=345989,790681,139065
BC01708=345989,790681,139065
BC01709=345989,790681,139065
BC01710=345989,790681,139065
BC01711=345989,790681,139065
BC01712=345989,790681,139065
BC01713=308625,748445,196549
BC01714=237635,668196,305769
BC01715=196160,672502,403752
BC01716=196160,672502,403752
BC01717=196160,727236,321537
BC01718=196160,765129,264619
BC01719=196160,765129,264619
BC01720=196160,765129,264619
BC01721=196160,765129,264619
BC01722=196160,765129,264619
BC01723=196160,765129,264619
BC01724=196160,765129,264619
BC01725=196160,765129,264619
BC01726=196160,765129,264619
BC01727=196160,765129,264619
BC01728=172117,778418,210988
BC01729=172117,778418,210988
BC01730=172117,778418,210988
BC01731=172117,778418,210988
BC01732=172117,778418,210988
BC01733=172117,778418,210988
BC01734=172117,778418,210988
BC01735=172117,778418,210988
BC01736=172117,778418,210988
BC01737=149065,790681,133702
BC01738=149065,790681,133702
BC01739=149065,790681,133702
BC01740=149065,790681,133702
BC01741=149065,790681,133702
BC01742=149065,790681,133702
BC01743=149065,790681,133702
BC01744=149065,790681,133702
BC01745=149065,790681,133702
BC01746=149065,790681,133702
BC01747=149065,790681,133702
BC01748=149065,790681,133702
BC01749=117513,790681,53
BC01750=117513,790681,53
BC01751=117513,790681,53
BC01752=117513,790681,53
BC01753=117513,790681,53
BC01754=117513,790681,53
BC01755=117513,790681,53
BC01756=117513,790681,53
BC01757=117513,790681,53
BC01758=117513,790681,53
BC01759=117513,790681,53
BC01760=117513,790681,53
BC01761=117513,790681,53
BC01762=190612,790681,158488
BC01763=190612,790681,158488
BC01764=190612,790681,158488
BC01765=190612,790681,158488
BC01766=190612,790681,158488
BC01767=190612,790681,158488
BC01768=184906,790681,111068
BC01769=184906,790681,111068
BC01770=184906,790681,111068
BC01771=184906,790681,111068
BC01772=184906,790681,111068
BC01773=184906,790681,111068
BC01774=181347,790681,153019
BC01775=174520,790681,233505
BC01776=174520,790681,233505
BC01777=174520,790681,233505
BC01778=174520,790681,233505
BC01779=174520,790681,233505
BC01780=174520,790681,233505
BC01781=184991,733498,315883
BC01782=196160,672502,403752
BC01783=196160,672502,403752
BC01784=237635,668196,305769
BC01785=308625,748445,196549
BC01786=309549,790681,184299
BC01787=309549,790681,184299
BC01788=309549,790681,184299
BC01789=309549,790681,184299
BC01790=309549,790681,184299
BC01791=309549,790681,184299
BC01792=321199,790681,207159
BC01793=321199,790681,207159
BC01794=321199,790681,207159
BC01795=321199,790681,207159
BC01796=321199,790681,207159
BC01797=321199,790681,207159
BC01798=321199,790681,207159
BC01799=321199,790681,207159
BC01800=373020,790681,107875
BC01801=373020,790681,107875
BC01802=373020,790681,107875
BC01803=373020,790681,107875
BC01804=373020,790681,107875
BC01805=373020,790681,107875
BC01806=373020,790681,107875
BC01807=373020,790681,107875
BC01808=367447,763418,217217
BC01809=362764,784495,185132
BC01810=361390,790681,53
BC01811=361390,790681,53
BC01812=361390,790681,53
BC01813=361390,790681,53
BC01814=361390,790681,53
BC01815=361390,790681,53
BC01816=340769,790681,53
BC01817=340769,790681,53
BC01818=340769,790681,53
BC01819=340769,790681,53
BC01820=340769,790681,53
BC01821=340769,790681,53
BC01822=340769,790681,53
BC01823=340769,790681,53
BC01824=340769,790681,53
BC01825=340769,790681,53
BC01826=340769,790681,53
BC01827=340769,790681,53
BC01828=340769,790681,53
BC01829=340769,790681,53
BC01830=340769,790681,53
BC01831=340769,765105,53
BC01832=340769,765105,53
BC01833=340769,765105,53
BC01834=340769,765105,53
BC01835=340769,765105,53
BC01836=340769,765105,53
BC01837=340769,765105,53
BC01838=326290,746662,147117
BC01839=300313,667687,410966
BC01840=300313,667687,410966
BC01841=200178,761203,279737
BC01842=168613,790681,238372
BC01843=168613,790681,238372
BC01844=168613,790681,238372
BC01845=168613,790681,238372
BC01846=168613,790681,238372
BC01847=168613,790681,238372
BC01848=187396,785580,192031
BC01849=187396,785580,192031
BC01850=187396,785580,192031
BC01851=187396,785580,192031
BC01852=187396,785580,192031
BC01853=187396,785580,192031
BC01854=200178,761203,279737
BC01855=300313,667687,410966
BC01856=300313,667687,410966
BC01857=326290,746662,147117
BC01858=326023,790681,196549
BC01859=326023,790681,196549
BC01860=326023,790681,196549
BC01861=326023,790681,196549
BC01862=326023,790681,196549
BC01863=326023,790681,196549
BC01864=316509,790681,152288
BC01865=316509,790681,152288
BC01866=316509,790681,152288
BC01867=316509,790681,152288
BC01868=316509,790681,152288
BC01869=316509,790681,152288
BC01870=314401,774670,185962
BC01871=300313,667687,410966
BC01872=300313,667687,410966
BC01873=200178,761203,279737
BC01874=186958,779092,256601
BC01875=178395,790681,241614
BC01876=178395,790681,241614
BC01877=178395,790681,241614
BC01878=178395,790681,241614
BC01879=178395,790681,241614
BC01880=178395,790681,241614
BC01881=198041,770354,161044
BC01882=198041,770354,161044
BC01883=198041,770354,161044
BC01884=198041,770354,161044
BC01885=198041,770354,161044
BC01886=198041,770354,161044
BC01887=200178,761203,279737
BC01888=300313,667687,410966
BC01889=300313,667687,410966
BC01890=363254,767093,179444
BC01891=378190,790681,124507
BC01892=378190,790681,124507
BC01893=378190,790681,124507
BC01894=378190,790681,124507
BC01895=378190,790681,124507
BC01896=378190,790681,124507
BC01897=345239,790681,222063
BC01898=345239,790681,222063
BC01899=345239,790681,222063
BC01900=345239,790681,222063
BC01901=345239,790681,222063
BC01902=345239,790681,222063
BC01903=363254,767093,179444
BC01904=300313,667687,410966
BC01905=300313,667687,410966
BC01906=200178,761203,279737
BC01907=142668,790681,138813
BC01908=142668,790681,138813
BC01909=142668,790681,138813
BC01910=142668,790681,138813
BC01911=142668,790681,138813
BC01912=142668,790681,138813
BC01913=142668,790681,138813
BC01914=142668,790681,138813
BC01915=203164,773756,23252
BC01916=203164,773756,23252
BC01917=203164,773756,23252
BC01918=203164,773756,23252
BC01919=203164,773756,23252
BC01920=203164,773756,23252
BC01921=200599,780936,88057
BC01922=197119,790681,176008
BC01923=197119,790681,176008
BC01924=197119,790681,176008
BC01925=197119,790681,176008
BC01926=197119,790681,176008
BC01927=197119,790681,176008
BC01928=197993,782258,205645
BC01929=199960,763308,272330
BC01930=201592,760202,280395
BC01931=200178,669563,279737
BC01932=78393,670967,1075175
EC00000=798156,0
EC00001=798153,3
EC00002=798156,0
EC00003=798156,0
EC00004=798156,0
EC00005=798156,0
EC00006=798156,0
EC00007=798156,0
EC00008=798156,0
EC00009=798156,0
EC00010=798156,0
EC00011=798156,0
EC00012=798156,0
EC00013=798156,0
EC00014=798156,0
EC00015=798156,0
EC00016=798156,0
EC00017=798156,0
EC00018=798156,0
EC00019=798156,0
EC00020=798156,0
EC00021=798156,0
EC00022=798154,2
EC00023=798154,2
EC00024=798154,2
EC00025=798154,2
EC00026=798154,2
EC00027=798154,2
EC00028=798154,2
EC00029=798156,0
EC00030=798156,0
EC00031=798156,0
EC00032=798156,0
EC00033=798156,0
EC00034=798156,0
EC00035=798156,0
EC00036=798156,0
EC00037=798156,0
EC00038=798156,0
EC00039=798156,0
EC00040=798156,0
EC00041=798156,0
EC00042=798156,0
EC00043=798156,0
EC00044=798156,0
EC00045=798156,0
EC00046=798156,0
EC00047=798156,0
EC00048=798156,0
EC00049=798156,0
EC00050=798156,0
EC00051=798156,0
EC00052=798156,0
EC00053=798156,0
EC00054=798156,0
EC00055=798156,0
EC00056=798156,0
EC00057=798156,0
EC00058=798156,0
EC00059=798156,0
EC00060=798156,0
EC00061=798156,0
EC00062=798156,0
EC00063=798156,0
EC00064=798156,0
EC00065=798156,0
EC00066=798156,0
EC00067=798156,0
EC00068=798156,0
EC00069=798156,0
EC00070=798156,0
EC00071=798156,0
EC00072=798156,0
EC00073=798156,0
EC00074=798156,0
EC00075=798156,0
EC00076=798156,0
EC00077=798156,0
EC00078=798156,0
EC00079=798156,0
EC00080=798156,0
EC00081=798156,0
EC00082=798156,0
EC00083=798156,0
EC00084=798156,0
EC00085=798156,0
EC00086=798156,0
EC00087=798156,0
EC00088=798156,0
EC00089=798156,0
EC00090=798156,0
EC00091=798156,0
EC00092=798156,0
EC00093=798156,0
EC00094=798156,0
EC00095=798156,0
EC00096=798156,0
EC00097=798156,0
EC00098=798156,0
EC00099=798156,0
EC00100=798156,0
EC00101=798156,0
EC00102=798156,0
EC00103=798156,0
EC00104=798156,0
EC00105=798156,0
EC00106=798156,0
EC00107=798156,0
EC00108=798156,0
EC00109=798156,0
EC00110=798156,0
EC00111=798156,0
EC00112=798156,0
EC00113=798156,0
EC00114=798156,0
EC00115=798156,0
EC00116=798156,0
EC00117=798156,0
EC00118=798156,0
EC00119=798156,0
EC00120=798156,0
EC00121=798156,0
EC00122=798155,0
EC00123=798155,0
EC00124=798155,0
EC00125=798155,0
EC00126=798155,0
EC00127=798155,0
EC00128=798155,0
EC00129=798155,0
EC00130=798155,0
EC00131=798156,0
EC00132=798156,0
EC00133=798156,0
EC00134=798155,1
EC00135=798155,1
EC00136=798155,1
EC00137=798155,1
EC00138=798155,1
EC00139=798155,1
EC00140=798155,1
EC00141=798155,1
EC00142=798156,0
EC00143=798156,0
EC00144=798156,0
EC00145=798156,0
EC00146=798156,0
EC00147=798156,0
EC00148=798156,0
EC00149=798156,0
EC00150=798156,0
EC00151=798156,0
EC00152=798156,0
EC00153=798156,0
EC00154=798156,0
EC00155=798156,0
EC00156=798156,0
EC00157=798156,0
EC00158=798156,0
EC00159=798156,0
EC00160=798156,0
EC00161=798156,0
EC00162=798156,0
EC00163=798156,0
EC00164=798156,0
EC00165=798156,0
EC00166=798156,0
EC00167=798156,0
EC00168=798156,0
EC00169=798156,0
EC00170=798156,0
EC00171=798156,0
EC00172=798156,0
EC00173=798156,0
EC00174=798156,0
EC00175=798156,0
EC00176=798156,0
EC00177=798156,0
EC00178=798156,0
EC00179=798156,0
EC00180=798156,0
EC00181=798156,0
EC00182=798156,0
EC00183=798156,0
EC00184=798156,0
EC00185=798156,0
EC00186=798156,0
EC00187=798155,0
EC00188=798155,0
EC00189=798155,0
EC00190=798155,0
EC00191=798155,0
EC00192=798155,0
EC00193=798155,0
EC00194=798155,0
EC00195=798155,0
EC00196=798153,2
EC00197=798156,0
EC00198=798156,0
EC00199=798156,0
EC00200=798156,0
EC00201=798156,0
EC00202=798156,0
EC00203=798156,0
EC00204=798156,0
EC00205=798156,0
EC00206=798156,0
EC00207=798156,0
EC00208=798156,0
EC00209=798156,0
EC00210=798156,0
EC00211=798156,0
EC00212=798156,0
EC00213=798156,0
EC00214=798156,0
EC00215=798156,0
EC00216=798156,0
EC00217=798156,0
EC00218=798156,0
EC00219=798156,0
EC00220=798156,0
EC00221=798156,0
EC00222=798156,0
EC00223=798156,0
EC00224=798156,0
EC00225=798156,0
EC00226=798156,0
EC00227=798156,0
EC00228=798156,0
EC00229=798156,0
EC00230=798156,0
EC00231=798156,0
EC00232=798155,0
EC00233=798155,0
EC00234=798155,0
EC00235=798155,0
EC00236=798155,0
EC00237=798155,0
EC00238=798155,0
EC00239=798155,0
EC00240=798155,0
EC00241=798156,0
EC00242=798155,0
EC00243=798155,0
EC00244=798154,1
EC00245=798154,1
EC00246=798154,1
EC00247=798154,1
EC00248=798154,1
EC00249=798154,1
EC00250=798154,1
EC00251=798154,1
EC00252=798154,1
EC00253=798156,0
EC00254=798156,0
EC00255=798156,0
EC00256=798156,0
EC00257=798156,0
EC00258=798156,0
EC00259=798156,0
EC00260=798156,0
EC00261=798156,0
EC00262=798156,0
EC00263=798156,0
EC00264=798156,0
EC00265=798156,0
EC00266=798156,0
EC00267=798156,0
EC00268=798155,0
EC00269=798155,0
EC00270=798155,0
EC00271=798155,0
EC00272=798155,0
EC00273=798155,0
EC00274=798155,0
EC00275=798155,0
EC00276=798155,0
EC00277=798155,0
EC00278=798155,0
EC00279=798156,0
EC00280=798156,0
EC00281=798156,0
EC00282=798156,0
EC00283=798156,0
EC00284=798156,0
EC00285=798156,0
EC00286=798156,0
EC00287=798156,0
EC00288=798156,0
EC00289=798156,0
EC00290=798156,0
EC00291=798156,0
EC00292=798156,0
EC00293=798156,0
EC00294=798156,0
EC00295=798156,0
EC00296=798156,0
EC00297=798156,0
EC00298=798156,0
EC00299=798156,0
EC00300=798156,0
EC00301=798156,0
EC00302=798156,0
EC00303=798156,0
EC00304=798156,0
EC00305=798156,0
EC00306=798156,0
EC00307=798156,0
EC00308=798156,0
EC00309=798154,2
EC00310=798156,0
EC00311=798156,0
EC00312=798156,0
EC00313=798156,0
EC00314=798156,0
EC00315=798156,0
EC00316=798156,0
EC00317=798156,0
EC00318=798156,0
EC00319=798156,0
EC00320=798156,0
EC00321=798156,0
EC00322=798156,0
EC00323=798156,-30
EC00324=798156,-30
EC00325=798156,-30
EC00326=798156,-30
EC00327=798156,-30
EC00328=798156,-30
EC00329=798156,-30
EC00330=798156,-30
EC00331=798156,-30
EC00332=798156,-30
EC00333=798156,-30
EC00334=798156,-28
EC00335=798156,0
EC00336=798156,0
EC00337=798156,0
EC00338=798156,0
EC00339=798156,0
EC00340=798156,0
EC00341=798156,0
EC00342=798156,0
EC00343=798156,0
EC00344=798156,0
EC00345=798156,0
EC00346=798156,0
EC00347=798156,0
EC00348=798156,0
EC00349=798156,0
EC00350=798156,0
EC00351=798156,0
EC00352=798156,0
EC00353=798156,0
EC00354=798156,0
EC00355=798156,0
EC00356=798156,0
EC00357=798156,0
EC00358=798156,0
EC00359=798156,0
EC00360=798156,0
EC00361=798156,0
EC00362=798156,0
EC00363=798156,0
EC00364=798156,0
EC00365=798156,0
EC00366=798156,0
EC00367=798156,0
EC00368=798156,0
EC00369=798156,0
EC00370=798156,0
EC00371=798156,0
EC00372=798156,0
EC00373=798156,0
EC00374=798156,0
EC00375=798156,0
EC00376=798156,0
EC00377=798156,0
EC00378=798156,0
EC00379=798156,0
EC00380=798156,0
EC00381=798156,0
EC00382=798156,0
EC00383=798156,0
EC00384=798156,0
EC00385=798156,0
EC00386=798156,0
EC00387=798156,0
EC00388=798156,0
EC00389=798156,0
EC00390=798156,0
EC00391=798156,0
EC00392=798156,0
EC00393=798156,0
EC00394=798156,0
EC00395=798156,0
EC00396=798156,0
EC00397=798156,0
EC00398=798156,0
EC00399=798156,0
EC00400=798156,0
EC00401=798156,0
EC00402=798156,0
EC00403=798156,0
EC00404=798156,0
EC00405=798156,0
EC00406=798156,0
EC00407=798156,0
EC00408=798156,0
EC00409=798156,0
EC00410=798156,0
EC00411=798156,0
EC00412=798156,0
EC00413=798156,0
EC00414=798156,0
EC00415=798156,0
EC00416=798156,0
EC00417=798156,0
EC00418=798156,0
EC00419=798156,0
EC00420=798156,0
EC00421=798156,0
EC00422=798156,0
EC00423=798156,0
EC00424=798156,0
EC00425=798156,0
EC00426=798156,0
EC00427=798156,0
EC00428=798156,0
EC00429=798156,0
EC00430=798156,0
EC00431=798156,0
EC00432=798156,0
EC00433=798156,0
EC00434=798156,0
EC00435=798156,0
EC00436=798156,0
EC00437=798156,0
EC00438=798156,0
EC00439=798156,0
EC00440=798156,0
EC00441=798156,0
EC00442=798156,0
EC00443=798156,0
EC00444=798156,0
EC00445=798156,0
EC00446=798156,0
EC00447=798156,0
EC00448=798156,0
EC00449=798156,0
EC00450=798156,0
EC00451=798156,0
EC00452=798156,0
EC00453=798156,0
EC00454=798156,0
EC00455=798156,0
EC00456=798156,0
EC00457=798156,0
EC00458=798156,0
EC00459=798156,0
EC00460=798156,0
EC00461=798156,0
EC00462=798156,0
EC00463=798156,0
EC00464=798156,0
EC00465=798156,0
EC00466=798156,0
EC00467=798156,0
EC00468=798156,0
EC00469=798156,0
EC00470=798156,0
EC00471=798156,0
EC00472=798156,0
EC00473=798156,0
EC00474=798140,8
EC00475=798155,0
EC00476=798156,0
EC00477=798156,0
EC00478=798156,0
EC00479=798156,0
EC00480=798154,0
EC00481=798154,0
EC00482=798156,0
EC00483=798156,0
EC00484=798156,0
EC00485=798156,0
EC00486=798156,0
EC00487=798156,0
EC00488=798156,0
EC00489=798156,0
EC00490=798156,0
EC00491=798156,0
EC00492=798156,0
EC00493=798156,0
EC00494=798156,0
EC00495=798156,0
EC00496=798156,0
EC00497=798156,0
EC00498=798156,0
EC00499=798156,0
EC00500=798156,0
EC00501=798156,0
EC00502=798156,0
EC00503=798156,0
EC00504=798156,0
EC00505=798156,0
EC00506=798156,0
EC00507=798156,0
EC00508=798155,0
EC00509=798155,0
EC00510=798156,0
EC00511=798155,0
EC00512=798156,0
EC00513=798156,0
EC00514=798156,0
EC00515=798156,0
EC00516=798156,0
EC00517=798156,0
EC00518=798156,0
EC00519=798156,0
EC00520=798156,0
EC00521=798156,0
EC00522=798156,0
EC00523=798156,0
EC00524=798156,0
EC00525=798156,0
EC00526=798156,0
EC00527=798156,0
EC00528=798156,0
EC00529=798156,0
EC00530=798156,0
EC00531=798156,0
EC00532=798156,0
EC00533=798156,0
EC00534=798156,0
EC00535=798156,0
EC00536=798156,0
EC00537=798156,0
EC00538=798156,0
EC00539=798156,0
EC00540=798156,0
EC00541=798156,0
EC00542=798156,0
EC00543=798156,0
EC00544=798155,1
EC00545=798155,1
EC00546=798156,0
EC00547=798156,0
EC00548=798156,0
EC00549=798156,0
EC00550=798156,0
EC00551=798156,0
EC00552=798156,0
EC00553=798156,0
EC00554=798156,0
EC00555=798156,0
EC00556=798156,0
EC00557=798156,0
EC00558=798156,0
EC00559=798156,0
EC00560=798156,0
EC00561=798156,0
EC00562=798156,0
EC00563=798156,0
EC00564=798156,0
EC00565=798154,1
EC00566=798154,1
EC00567=798154,1
EC00568=798154,1
EC00569=798151,2
EC00570=798156,0
EC00571=798156,0
EC00572=798156,0
EC00573=798156,0
EC00574=798156,0
EC00575=798156,0
EC00576=798156,0
EC00577=798156,0
EC00578=798156,0
EC00579=798156,0
EC00580=798156,0
EC00581=798156,0
EC00582=798156,0
EC00583=798156,0
EC00584=798156,0
EC00585=798156,0
EC00586=798156,0
EC00587=798156,0
EC00588=798156,0
EC00589=798156,0
EC00590=798156,0
EC00591=798156,0
EC00592=798156,0
EC00593=798156,0
EC00594=798156,0
EC00595=798156,0
EC00596=798156,0
EC00597=798156,0
EC00598=798156,0
EC00599=798156,0
EC00600=798156,0
EC00601=798156,0
EC00602=798156,0
EC00603=798156,0
EC00604=798156,0
EC00605=798156,0
EC00606=798156,0
EC00607=798156,0
EC00608=798156,0
EC00609=798156,0
EC00610=798156,0
EC00611=798156,0
EC00612=798156,0
EC00613=798156,0
EC00614=798156,0
EC00615=798156,0
EC00616=798156,0
EC00617=798156,0
EC00618=798156,0
EC00619=798156,0
EC00620=798156,0
EC00621=798156,0
EC00622=798156,0
EC00623=798156,0
EC00624=798156,0
EC00625=798156,0
EC00626=798156,0
EC00627=798156,0
EC00628=798155,1
EC00629=798155,1
EC00630=798156,0
EC00631=798156,0
EC00632=798156,0
EC00633=798156,0
EC00634=798156,0
EC00635=798156,0
EC00636=798156,0
EC00637=798156,0
EC00638=798156,0
EC00639=798156,0
EC00640=798156,0
EC00641=798156,0
EC00642=798156,0
EC00643=798156,0
EC00644=798156,0
EC00645=798156,0
EC00646=798156,0
EC00647=798156,0
EC00648=798156,0
EC00649=798156,0
EC00650=798156,0
EC00651=798156,0
EC00652=798156,0
EC00653=798156,0
EC00654=798156,0
EC00655=798156,0
EC00656=798156,0
EC00657=798156,0
EC00658=798156,0
EC00659=798156,0
EC00660=798156,0
EC00661=798156,0
EC00662=798156,0
EC00663=798156,0
EC00664=798156,0
EC00665=798156,0
EC00666=798156,0
EC00667=798156,1
EC00668=798156,0
EC00669=798156,0
EC00670=798156,0
EC00671=798156,0
EC00672=798156,0
EC00673=798156,0
EC00674=798156,0
EC00675=798156,0
EC00676=798156,0
EC00677=798156,0
EC00678=798156,0
EC00679=798156,0
EC00680=798156,0
EC00681=798156,0
EC00682=798156,0
EC00683=798156,0
EC00684=798156,0
EC00685=798156,0
EC00686=798156,0
EC00687=798156,0
EC00688=798156,0
EC00689=798156,0
EC00690=798156,0
EC00691=798156,0
EC00692=798156,0
EC00693=798156,0
EC00694=798156,0
EC00695=798156,0
EC00696=798156,0
EC00697=798155,1
EC00698=798155,1
EC00699=798155,1
EC00700=798156,0
EC00701=798156,0
EC00702=798156,0
EC00703=798156,0
EC00704=798156,0
EC00705=798156,0
EC00706=798156,0
EC00707=798156,0
EC00708=798156,0
EC00709=798156,0
EC00710=798156,0
EC00711=798156,0
EC00712=798156,0
EC00713=798156,0
EC00714=798156,0
EC00715=798156,0
EC00716=798156,0
EC00717=798156,0
EC00718=798156,0
EC00719=798156,0
EC00720=798156,0
EC00721=798156,0
EC00722=798156,0
EC00723=798156,0
EC00724=798156,0
EC00725=798156,0
EC00726=798156,0
EC00727=798156,0
EC00728=798156,0
EC00729=798156,0
EC00730=798156,0
EC00731=798156,0
EC00732=798156,0
EC00733=798156,0
EC00734=798156,0
EC00735=798156,0
EC00736=798156,0
EC00737=798156,0
EC00738=798156,0
EC00739=798156,0
EC00740=798156,0
EC00741=798156,0
EC00742=798156,0
EC00743=798156,0
EC00744=798156,0
EC00745=798156,0
EC00746=798156,0
EC00747=798156,0
EC00748=798156,0
EC00749=798156,0
EC00750=798156,0
EC00751=798156,0
EC00752=798156,0
EC00753=798156,0
EC00754=798156,0
EC00755=798156,0
EC00756=798156,0
EC00757=798156,0
EC00758=798156,0
EC00759=798156,0
EC00760=798156,0
EC00761=798156,0
EC00762=798156,0
EC00763=798155,0
EC00764=798156,0
EC00765=798156,0
EC00766=798156,0
EC00767=798156,0
EC00768=798155,1
EC00769=798155,1
EC00770=798155,1
EC00771=798156,0
EC00772=798156,0
EC00773=798156,0
EC00774=798156,0
EC00775=798156,0
EC00776=798156,0
EC00777=798156,0
EC00778=798156,0
EC00779=798156,0
EC00780=798156,0
EC00781=798155,0
EC00782=798156,0
EC00783=798156,0
EC00784=798156,0
EC00785=798156,0
EC00786=798156,0
EC00787=798156,0
EC00788=798155,1
EC00789=798156,0
EC00790=798156,1
EC00791=798156,1
EC00792=798156,0
EC00793=798156,0
EC00794=798156,0
EC00795=798156,0
EC00796=798156,0
EC00797=798156,0
EC00798=798156,0
EC00799=798156,0
EC00800=798156,0
EC00801=798156,0
EC00802=798156,0
EC00803=798156,0
EC00804=798156,0
EC00805=798156,0
EC00806=798156,0
EC00807=798156,0
EC00808=798155,0
EC00809=798156,0
EC00810=798156,0
EC00811=798156,0
EC00812=798156,0
EC00813=798156,0
EC00814=798156,0
EC00815=798156,0
EC00816=798156,0
EC00817=798156,0
EC00818=798156,0
EC00819=798156,0
EC00820=798156,0
EC00821=798156,0
EC00822=798156,0
EC00823=798156,0
EC00824=798156,0
EC00825=798156,0
EC00826=798156,0
EC00827=798156,0
EC00828=798156,0
EC00829=798156,0
EC00830=798156,0
EC00831=798156,0
EC00832=798156,0
EC00833=798156,0
EC00834=798156,0
EC00835=798156,0
EC00836=798156,0
EC00837=798156,0
EC00838=798156,0
EC00839=798156,0
EC00840=798156,0
EC00841=798156,0
EC00842=798156,0
EC00843=798156,0
EC00844=798156,0
EC00845=798156,0
EC00846=798156,0
EC00847=798156,0
EC00848=798156,0
EC00849=798156,0
EC00850=798156,0
EC00851=798156,0
EC00852=798156,0
EC00853=798156,0
EC00854=798156,0
EC00855=798156,0
EC00856=798156,0
EC00857=798156,0
EC00858=798156,0
EC00859=798156,0
EC00860=798156,0
EC00861=798156,0
EC00862=798156,0
EC00863=798156,0
EC00864=798156,0
EC00865=798156,0
EC00866=798156,0
EC00867=798156,0
EC00868=798153,2
EC00869=798153,2
EC00870=798153,2
EC00871=798153,2
EC00872=798153,2
EC00873=798153,2
EC00874=798153,2
EC00875=798153,2
EC00876=798152,2
EC00877=798152,2
EC00878=798152,2
EC00879=798152,2
EC00880=798152,2
EC00881=798152,2
EC00882=798152,2
EC00883=798153,1
EC00884=798156,0
EC00885=798156,0
EC00886=798153,3
EC00887=798156,0
EC00888=798156,0
EC00889=798156,0
EC00890=798156,0
EC00891=798156,0
EC00892=798156,0
EC00893=798156,0
EC00894=798156,0
EC00895=798156,0
EC00896=798156,0
EC00897=798156,0
EC00898=798156,0
EC00899=798156,0
EC00900=798156,0
EC00901=798156,0
EC00902=798156,0
EC00903=798156,0
EC00904=798156,0
EC00905=798156,0
EC00906=798156,0
EC00907=798156,0
EC00908=798156,0
EC00909=798156,0
EC00910=798156,0
EC00911=798156,0
EC00912=798156,0
EC00913=798156,0
EC00914=798156,0
EC00915=798156,0
EC00916=798156,0
EC00917=798156,0
EC00918=798156,0
EC00919=798156,0
EC00920=798156,0
EC00921=798156,0
EC00922=798156,0
EC00923=798156,0
EC00924=798156,0
EC00925=798156,0
EC00926=798156,0
EC00927=798156,0
EC00928=798156,0
EC00929=798156,0
EC00930=798156,0
EC00931=798156,0
EC00932=798156,0
EC00933=798156,0
EC00934=798156,0
EC00935=798156,0
EC00936=798156,0
EC00937=798156,0
EC00938=798156,0
EC00939=798156,0
EC00940=798156,0
EC00941=798156,0
EC00942=798156,0
EC00943=798156,0
EC00944=798156,0
EC00945=798156,0
EC00946=798156,0
EC00947=798156,0
EC00948=798156,0
EC00949=798156,0
EC00950=798156,0
EC00951=798156,0
EC00952=798156,0
EC00953=798156,0
EC00954=798156,0
EC00955=798156,0
EC00956=798156,0
EC00957=798156,0
EC00958=798156,0
EC00959=798156,0
EC00960=798156,0
EC00961=798156,0
EC00962=798156,0
EC00963=798156,0
EC00964=798156,0
EC00965=798156,0
EC00966=798156,0
EC00967=798156,0
EC00968=798156,0
EC00969=798156,0
EC00970=798156,0
EC00971=798156,0
EC00972=798156,0
EC00973=798156,0
EC00974=798156,0
EC00975=798156,0
EC00976=798156,0
EC00977=798156,0
EC00978=798156,0
EC00979=798156,0
EC00980=798156,0
EC00981=798156,0
EC00982=798156,0
EC00983=798156,0
EC00984=798156,0
EC00985=798156,0
EC00986=798156,0
EC00987=798156,0
EC00988=798156,0
EC00989=798156,0
EC00990=798156,0
EC00991=798156,0
EC00992=798156,0
EC00993=798156,0
EC00994=798156,0
EC00995=798156,0
EC00996=798156,0
EC00997=798156,0
EC00998=798156,0
EC00999=798156,0
EC01000=798155,0
EC01001=798155,0
EC01002=798155,0
EC01003=798155,0
EC01004=798155,0
EC01005=798155,0
EC01006=798155,0
EC01007=798155,0
EC01008=798155,0
EC01009=798156,0
EC01010=798156,0
EC01011=798156,0
EC01012=798156,0
EC01013=798156,0
EC01014=798156,0
EC01015=798156,0
EC01016=798156,0
EC01017=798156,0
EC01018=798156,0
EC01019=798156,0
EC01020=798156,0
EC01021=798156,0
EC01022=798156,0
EC01023=798156,0
EC01024=798156,0
EC01025=798156,0
EC01026=798156,0
EC01027=798156,0
EC01028=798156,0
EC01029=798156,0
EC01030=798156,0
EC01031=798156,0
EC01032=798156,0
EC01033=798156,0
EC01034=798156,0
EC01035=798156,0
EC01036=798156,0
EC01037=798156,0
EC01038=798156,0
EC01039=798156,0
EC01040=798156,0
EC01041=798156,0
EC01042=798156,0
EC01043=798156,0
EC01044=798156,0
EC01045=798156,0
EC01046=798156,0
EC01047=798156,0
EC01048=798156,0
EC01049=798156,0
EC01050=798156,0
EC01051=798156,0
EC01052=798156,0
EC01053=798156,0
EC01054=798156,0
EC01055=798156,0
EC01056=798156,0
EC01057=798156,0
EC01058=798156,0
EC01059=798156,0
EC01060=798156,0
EC01061=798156,0
EC01062=798156,0
EC01063=798156,0
EC01064=798156,0
EC01065=798156,0
EC01066=798156,0
EC01067=798156,0
EC01068=798156,0
EC01069=798156,0
EC01070=798156,0
EC01071=798156,0
EC01072=798156,0
EC01073=798156,0
EC01074=798156,0
EC01075=798156,0
EC01076=798156,0
EC01077=798156,0
EC01078=798156,0
EC01079=798156,0
EC01080=798156,0
EC01081=798156,0
EC01082=798156,0
EC01083=798156,0
EC01084=798156,0
EC01085=798156,0
EC01086=798156,0
EC01087=798156,0
EC01088=798156,0
EC01089=798156,0
EC01090=798156,0
EC01091=798156,0
EC01092=798156,0
EC01093=798156,0
EC01094=798156,0
EC01095=798156,0
EC01096=798156,0
EC01097=798156,0
EC01098=798156,0
EC01099=798156,0
EC01100=798156,0
EC01101=798156,0
EC01102=798156,0
EC01103=798156,0
EC01104=798156,0
EC01105=798156,0
EC01106=798156,0
EC01107=798156,0
EC01108=798156,0
EC01109=798156,0
EC01110=798156,0
EC01111=798156,0
EC01112=798156,0
EC01113=798156,0
EC01114=798156,0
EC01115=798156,0
EC01116=798156,0
EC01117=798156,0
EC01118=798156,0
EC01119=798156,0
EC01120=798156,0
EC01121=798156,0
EC01122=798156,0
EC01123=798156,0
EC01124=798156,0
EC01125=798156,0
EC01126=798156,0
EC01127=798156,0
EC01128=798154,2
EC01129=798156,0
EC01130=798156,0
EC01131=798156,0
EC01132=798156,0
EC01133=798156,0
EC01134=798156,0
EC01135=798156,0
EC01136=798156,0
EC01137=798156,0
EC01138=798156,0
EC01139=798156,0
EC01140=798156,0
EC01141=798156,0
EC01142=798156,0
EC01143=798156,0
EC01144=798156,0
EC01145=798156,0
EC01146=798156,0
EC01147=798156,0
EC01148=798156,0
EC01149=798156,0
EC01150=798156,0
EC01151=798156,0
EC01152=798156,0
EC01153=798156,0
EC01154=798156,0
EC01155=798156,0
EC01156=798156,0
EC01157=798156,0
EC01158=798156,0
EC01159=798156,0
EC01160=798156,0
EC01161=798156,0
EC01162=798156,0
EC01163=798156,0
EC01164=798156,0
EC01165=798156,0
EC01166=798156,0
EC01167=798156,0
EC01168=798156,0
EC01169=798156,0
EC01170=798156,0
EC01171=798156,0
EC01172=798156,0
EC01173=798156,0
EC01174=798156,0
EC01175=798156,0
EC01176=798156,0
EC01177=798156,0
EC01178=798156,0
EC01179=798156,0
EC01180=798156,0
EC01181=798156,0
EC01182=798156,0
EC01183=798156,0
EC01184=798156,0
EC01185=798156,0
EC01186=798156,0
EC01187=798156,0
EC01188=798156,0
EC01189=798156,0
EC01190=798156,0
EC01191=798156,0
EC01192=798156,0
EC01193=798156,0
EC01194=798156,0
EC01195=798156,0
EC01196=798156,0
EC01197=798156,0
EC01198=798156,0
EC01199=798156,0
EC01200=798156,0
EC01201=798156,0
EC01202=798156,0
EC01203=798156,0
EC01204=798156,0
EC01205=798156,0
EC01206=798156,0
EC01207=798156,0
EC01208=798156,0
EC01209=798156,0
EC01210=798156,0
EC01211=798156,0
EC01212=798156,0
EC01213=798156,0
EC01214=798156,0
EC01215=798156,0
EC01216=798156,0
EC01217=798156,0
EC01218=798156,0
EC01219=798156,0
EC01220=798156,0
EC01221=798156,0
EC01222=798156,0
EC01223=798156,0
EC01224=798156,0
EC01225=798156,0
EC01226=798156,0
EC01227=798156,0
EC01228=798156,0
EC01229=798156,0
EC01230=798156,0
EC01231=798156,0
EC01232=798156,0
EC01233=798156,0
EC01234=798156,0
EC01235=798156,0
EC01236=798156,0
EC01237=798156,0
EC01238=798156,0
EC01239=798156,0
EC01240=798156,0
EC01241=798156,0
EC01242=798156,0
EC01243=798156,0
EC01244=798156,0
EC01245=798156,0
EC01246=798156,0
EC01247=798156,0
EC01248=798156,0
EC01249=798156,0
EC01250=798156,0
EC01251=798156,0
EC01252=798156,0
EC01253=798156,0
EC01254=798156,0
EC01255=798156,0
EC01256=798156,0
EC01257=798156,0
EC01258=798156,0
EC01259=798140,8
EC01260=798155,0
EC01261=798156,0
EC01262=798156,0
EC01263=798156,0
EC01264=798156,0
EC01265=798154,0
EC01266=798154,0
EC01267=798156,0
EC01268=798156,0
EC01269=798156,0
EC01270=798156,0
EC01271=798156,0
EC01272=798156,0
EC01273=798156,0
EC01274=798156,0
EC01275=798156,0
EC01276=798156,0
EC01277=798156,0
EC01278=798156,0
EC01279=798156,0
EC01280=798156,0
EC01281=798156,0
EC01282=798156,0
EC01283=798156,0
EC01284=798156,0
EC01285=798156,0
EC01286=798156,0
EC01287=798156,0
EC01288=798156,0
EC01289=798156,0
EC01290=798156,0
EC01291=798156,0
EC01292=798156,0
EC01293=798155,0
EC01294=798155,0
EC01295=798156,0
EC01296=798155,0
EC01297=798156,0
EC01298=798156,0
EC01299=798156,0
EC01300=798156,0
EC01301=798156,0
EC01302=798156,0
EC01303=798156,0
EC01304=798156,0
EC01305=798156,0
EC01306=798156,0
EC01307=798156,0
EC01308=798156,0
EC01309=798156,0
EC01310=798156,0
EC01311=798156,0
EC01312=798156,0
EC01313=798156,0
EC01314=798156,0
EC01315=798156,0
EC01316=798156,0
EC01317=798156,0
EC01318=798156,0
EC01319=798156,0
EC01320=798156,0
EC01321=798156,0
EC01322=798156,0
EC01323=798156,0
EC01324=798156,0
EC01325=798156,0
EC01326=798156,0
EC01327=798156,0
EC01328=798156,0
EC01329=798156,0
EC01330=798156,0
EC01331=798156,0
EC01332=798156,0
EC01333=798156,0
EC01334=798156,0
EC01335=798156,0
EC01336=798156,0
EC01337=798156,0
EC01338=798156,0
EC01339=798156,0
EC01340=798156,0
EC01341=798156,0
EC01342=798156,0
EC01343=798156,0
EC01344=798156,0
EC01345=798154,1
EC01346=798154,1
EC01347=798154,1
EC01348=798154,1
EC01349=798151,2
EC01350=798156,0
EC01351=798156,0
EC01352=798156,0
EC01353=798156,0
EC01354=798156,0
EC01355=798156,0
EC01356=798156,0
EC01357=798156,0
EC01358=798156,0
EC01359=798156,0
EC01360=798156,0
EC01361=798156,0
EC01362=798156,0
EC01363=798156,0
EC01364=798156,0
EC01365=798156,0
EC01366=798156,0
EC01367=798156,0
EC01368=798156,0
EC01369=798156,0
EC01370=798156,0
EC01371=798156,0
EC01372=798156,0
EC01373=798156,0
EC01374=798156,0
EC01375=798156,0
EC01376=798156,0
EC01377=798156,0
EC01378=798156,0
EC01379=798156,0
EC01380=798156,0
EC01381=798156,0
EC01382=798156,0
EC01383=798156,0
EC01384=798156,0
EC01385=798156,0
EC01386=798156,0
EC01387=798156,0
EC01388=798156,0
EC01389=798156,0
EC01390=798156,0
EC01391=798156,0
EC01392=798156,0
EC01393=798156,0
EC01394=798156,0
EC01395=798156,0
EC01396=798156,0
EC01397=798156,0
EC01398=798156,0
EC01399=798156,0
EC01400=798156,0
EC01401=798156,0
EC01402=798156,0
EC01403=798156,0
EC01404=798156,0
EC01405=798156,0
EC01406=798156,0
EC01407=798156,0
EC01408=798156,0
EC01409=798156,0
EC01410=798156,0
EC01411=798156,0
EC01412=798156,0
EC01413=798156,0
EC01414=798156,0
EC01415=798156,0
EC01416=798156,0
EC01417=798156,0
EC01418=798156,0
EC01419=798156,0
EC01420=798156,0
EC01421=798156,0
EC01422=798156,0
EC01423=798156,0
EC01424=798156,0
EC01425=798156,0
EC01426=798156,0
EC01427=798156,0
EC01428=798156,0
EC01429=798156,0
EC01430=798156,0
EC01431=798156,0
EC01432=798156,0
EC01433=798156,0
EC01434=798156,0
EC01435=798156,0
EC01436=798156,0
EC01437=798156,0
EC01438=798156,0
EC01439=798156,0
EC01440=798156,0
EC01441=798156,1
EC01442=798156,0
EC01443=798156,0
EC01444=798156,0
EC01445=798156,0
EC01446=798156,0
EC01447=798156,0
EC01448=798156,0
EC01449=798156,0
EC01450=798156,0
EC01451=798156,0
EC01452=798156,0
EC01453=798156,0
EC01454=798156,0
EC01455=798156,0
EC01456=798156,0
EC01457=798156,0
EC01458=798156,0
EC01459=798156,0
EC01460=798156,0
EC01461=798156,0
EC01462=798156,0
EC01463=798156,0
EC01464=798156,0
EC01465=798156,0
EC01466=798156,0
EC01467=798156,0
EC01468=798156,0
EC01469=798156,0
EC01470=798156,0
EC01471=798156,0
EC01472=798156,0
EC01473=798156,0
EC01474=798156,0
EC01475=798156,0
EC01476=798156,0
EC01477=798156,0
EC01478=798156,0
EC01479=798156,0
EC01480=798156,0
EC01481=798156,0
EC01482=798156,0
EC01483=798156,0
EC01484=798156,0
EC01485=798156,0
EC01486=798156,0
EC01487=798156,0
EC01488=798156,0
EC01489=798156,0
EC01490=798156,0
EC01491=798156,0
EC01492=798156,0
EC01493=798156,0
EC01494=798156,0
EC01495=798156,0
EC01496=798156,0
EC01497=798156,0
EC01498=798156,0
EC01499=798156,0
EC01500=798156,0
EC01501=798156,0
EC01502=798156,0
EC01503=798156,0
EC01504=798156,0
EC01505=798156,0
EC01506=798156,0
EC01507=798156,0
EC01508=798156,0
EC01509=798156,0
EC01510=798156,0
EC01511=798156,0
EC01512=798156,0
EC01513=798156,0
EC01514=798156,0
EC01515=798156,0
EC01516=798156,0
EC01517=798156,0
EC01518=798156,0
EC01519=798156,0
EC01520=798156,0
EC01521=798156,0
EC01522=798156,0
EC01523=798156,0
EC01524=798156,0
EC01525=798156,0
EC01526=798156,0
EC01527=798156,0
EC01528=798156,0
EC01529=798156,0
EC01530=798156,0
EC01531=798156,0
EC01532=798156,0
EC01533=798156,0
EC01534=798155,0
EC01535=798156,0
EC01536=798156,0
EC01537=798156,0
EC01538=798156,0
EC01539=798155,1
EC01540=798155,1
EC01541=798155,1
EC01542=798156,0
EC01543=798156,0
EC01544=798156,0
EC01545=798156,0
EC01546=798156,0
EC01547=798156,0
EC01548=798156,0
EC01549=798156,0
EC01550=798156,0
EC01551=798156,0
EC01552=798156,0
EC01553=798156,0
EC01554=798156,0
EC01555=798156,0
EC01556=798156,0
EC01557=798156,0
EC01558=798156,0
EC01559=798156,0
EC01560=798156,0
EC01561=798156,0
EC01562=798156,0
EC01563=798156,0
EC01564=798156,0
EC01565=798156,0
EC01566=798156,0
EC01567=798156,0
EC01568=798156,0
EC01569=798156,0
EC01570=798156,0
EC01571=798156,0
EC01572=798156,0
EC01573=798156,0
EC01574=798156,0
EC01575=798156,0
EC01576=798156,0
EC01577=798156,0
EC01578=798156,0
EC01579=798155,0
EC01580=798156,0
EC01581=798156,0
EC01582=798156,0
EC01583=798156,0
EC01584=798156,0
EC01585=798156,0
EC01586=798156,0
EC01587=798156,0
EC01588=798156,0
EC01589=798156,0
EC01590=798156,0
EC01591=798156,0
EC01592=798156,0
EC01593=798156,0
EC01594=798156,0
EC01595=798156,0
EC01596=798156,0
EC01597=798156,0
EC01598=798156,0
EC01599=798156,0
EC01600=798156,0
EC01601=798156,0
EC01602=798156,0
EC01603=798156,0
EC01604=798156,0
EC01605=798156,0
EC01606=798156,0
EC01607=798156,0
EC01608=798156,0
EC01609=798156,0
EC01610=798156,0
EC01611=798156,0
EC01612=798156,0
EC01613=798156,0
EC01614=798156,0
EC01615=798156,0
EC01616=798156,0
EC01617=798156,0
EC01618=798156,0
EC01619=798156,0
EC01620=798156,0
EC01621=798156,0
EC01622=798156,0
EC01623=798156,0
EC01624=798156,0
EC01625=798156,0
EC01626=798156,0
EC01627=798156,0
EC01628=798156,0
EC01629=798156,0
EC01630=798156,0
EC01631=798156,0
EC01632=798156,0
EC01633=798156,0
EC01634=798156,0
EC01635=798156,0
EC01636=798156,0
EC01637=798153,2
EC01638=798153,2
EC01639=798153,2
EC01640=798153,2
EC01641=798153,2
EC01642=798153,2
EC01643=798153,2
EC01644=798153,2
EC01645=798152,2
EC01646=798152,2
EC01647=798152,2
EC01648=798152,2
EC01649=798152,2
EC01650=798152,2
EC01651=798152,2
EC01652=798153,1
EC01653=798156,0
EC01654=798156,0
EC01655=798156,0
EC01656=798156,0
EC01657=798156,0
EC01658=798156,0
EC01659=798156,0
EC01660=798156,0
EC01661=798156,0
EC01662=798156,0
EC01663=798156,0
EC01664=798156,0
EC01665=798156,0
EC01666=798156,0
EC01667=798156,0
EC01668=798156,0
EC01669=798156,0
EC01670=798156,0
EC01671=798156,0
EC01672=798156,0
EC01673=798156,0
EC01674=798156,0
EC01675=798156,0
EC01676=798156,0
EC01677=798156,0
EC01678=798156,0
EC01679=798156,0
EC01680=798156,0
EC01681=798154,1
EC01682=798154,1
EC01683=798156,0
EC01684=798156,0
EC01685=798156,0
EC01686=798156,0
EC01687=798156,0
EC01688=798156,0
EC01689=798156,0
EC01690=798156,0
EC01691=798156,0
EC01692=798156,0
EC01693=798156,0
EC01694=798156,0
EC01695=798156,0
EC01696=798156,0
EC01697=798156,0
EC01698=798156,0
EC01699=798156,0
EC01700=798156,0
EC01701=798156,0
EC01702=798156,0
EC01703=798156,0
EC01704=798156,0
EC01705=798156,0
EC01706=798156,0
EC01707=798156,0
EC01708=798156,0
EC01709=798156,0
EC01710=798156,0
EC01711=798156,0
EC01712=798156,0
EC01713=798156,0
EC01714=798156,0
EC01715=798156,0
EC01716=798156,0
EC01717=798156,0
EC01718=798156,0
EC01719=798156,0
EC01720=798156,0
EC01721=798156,0
EC01722=798156,0
EC01723=798156,0
EC01724=798156,0
EC01725=798156,0
EC01726=798156,0
EC01727=798156,0
EC01728=798156,0
EC01729=798156,0
EC01730=798156,0
EC01731=798156,0
EC01732=798156,0
EC01733=798156,0
EC01734=798156,0
EC01735=798156,0
EC01736=798156,0
EC01737=798156,0
EC01738=798156,0
EC01739=798156,0
EC01740=798156,0
EC01741=798156,0
EC01742=798156,0
EC01743=798156,0
EC01744=798156,0
EC01745=798156,0
EC01746=798156,0
EC01747=798156,0
EC01748=798156,0
EC01749=798156,0
EC01750=798156,0
EC01751=798156,0
EC01752=798156,0
EC01753=798156,0
EC01754=798156,0
EC01755=798156,0
EC01756=798156,0
EC01757=798156,0
EC01758=798156,0
EC01759=798156,0
EC01760=798156,0
EC01761=798156,0
EC01762=798156,0
EC01763=798156,0
EC01764=798156,0
EC01765=798156,0
EC01766=798156,0
EC01767=798156,0
EC01768=798156,0
EC01769=798156,0
EC01770=798156,0
EC01771=798156,0
EC01772=798156,0
EC01773=798156,0
EC01774=798156,0
EC01775=798156,0
EC01776=798156,0
EC01777=798156,0
EC01778=798156,0
EC01779=798156,0
EC01780=798156,0
EC01781=798156,0
EC01782=798156,0
EC01783=798156,0
EC01784=798156,0
EC01785=798156,0
EC01786=798156,0
EC01787=798156,0
EC01788=798156,0
EC01789=798156,0
EC01790=798156,0
EC01791=798156,0
EC01792=798156,0
EC01793=798156,0
EC01794=798156,0
EC01795=798156,0
EC01796=798156,0
EC01797=798156,0
EC01798=798156,0
EC01799=798156,0
EC01800=798156,0
EC01801=798156,0
EC01802=798156,0
EC01803=798156,0
EC01804=798156,0
EC01805=798156,0
EC01806=798156,0
EC01807=798156,0
EC01808=798156,0
EC01809=798156,0
EC01810=798156,0
EC01811=798156,0
EC01812=798156,0
EC01813=798156,0
EC01814=798156,0
EC01815=798156,0
EC01816=798156,0
EC01817=798156,0
EC01818=798156,0
EC01819=798156,0
EC01820=798156,0
EC01821=798156,0
EC01822=798156,0
EC01823=798156,0
EC01824=798156,0
EC01825=798156,0
EC01826=798156,0
EC01827=798156,0
EC01828=798156,0
EC01829=798156,0
EC01830=798156,0
EC01831=798156,0
EC01832=798156,0
EC01833=798156,0
EC01834=798156,0
EC01835=798156,0
EC01836=798156,0
EC01837=798156,0
EC01838=798156,0
EC01839=798156,0
EC01840=798156,0
EC01841=798156,0
EC01842=798156,0
EC01843=798156,0
EC01844=798156,0
EC01845=798156,0
EC01846=798156,0
EC01847=798156,0
EC01848=798156,0
EC01849=798156,0
EC01850=798156,0
EC01851=798156,0
EC01852=798156,0
EC01853=798156,0
EC01854=798156,0
EC01855=798156,0
EC01856=798156,0
EC01857=798156,0
EC01858=798156,0
EC01859=798156,0
EC01860=798156,0
EC01861=798156,0
EC01862=798156,0
EC01863=798156,0
EC01864=798156,0
EC01865=798156,0
EC01866=798156,0
EC01867=798156,0
EC01868=798156,0
EC01869=798156,0
EC01870=798156,0
EC01871=798156,0
EC01872=798156,0
EC01873=798156,0
EC01874=798156,0
EC01875=798156,0
EC01876=798156,0
EC01877=798156,0
EC01878=798156,0
EC01879=798156,0
EC01880=798156,0
EC01881=798156,0
EC01882=798156,0
EC01883=798156,0
EC01884=798156,0
EC01885=798156,0
EC01886=798156,0
EC01887=798156,0
EC01888=798156,0
EC01889=798156,0
EC01890=798156,0
EC01891=798156,0
EC01892=798156,0
EC01893=798156,0
EC01894=798156,0
EC01895=798156,0
EC01896=798156,0
EC01897=798156,0
EC01898=798156,0
EC01899=798156,0
EC01900=798156,0
EC01901=798156,0
EC01902=798156,0
EC01903=798156,0
EC01904=798156,0
EC01905=798156,0
EC01906=798156,0
EC01907=798156,0
EC01908=798156,0
EC01909=798156,0
EC01910=798156,0
EC01911=798156,0
EC01912=798156,0
EC01913=798156,0
EC01914=798156,0
EC01915=798156,0
EC01916=798156,0
EC01917=798156,0
EC01918=798156,0
EC01919=798156,0
EC01920=798156,0
EC01921=798156,0
EC01922=798156,0
EC01923=798156,0
EC01924=798156,0
EC01925=798156,0
EC01926=798156,0
EC01927=798156,0
EC01928=798156,0
EC01929=798156,0
EC01930=798156,0
EC01931=798156,0
EC01932=798156,0
///POSTYPE BASE
///RECTAN
///RCONF 0,0,0,0,0,0,0,0,0,0,0,0,0,0,0,0,0,0,0,0,0,0,0,0
P00006=0.000,0.000,0.000,0.0000,0.0000,0.0000
P00021=3.198,-0.012,-3.236,0.0000,0.0000,0.0000
P00022=7.754,0.769,-4.150,0.0000,0.0000,0.0000
P00023=0.105,0.010,-3.143,0.0000,0.0000,0.0000
P00024=0.145,-0.552,1.326,0.0000,0.0000,0.0000
P00025=-2.003,0.006,0.728,0.0000,0.0000,0.0000
P00026=0.562,-0.002,-0.337,0.0000,0.0000,0.0000
P00027=-0.746,0.015,-9.096,0.0000,0.0000,0.0000
P00028=-2.237,-0.018,-7.702,0.0000,0.0000,0.0000
P00029=-2.156,-0.086,-4.681,0.0000,0.0000,0.0000
P00030=5.926,-4.294,-1.390,0.0000,0.0000,0.0000
P00031=1.853,-0.001,-1.549,0.0000,0.0000,0.0000
P00032=1.957,0.503,-7.217,0.0000,0.0000,0.0000
///RCONF 0,0,0,0,1,0,0,0,0,0,0,0,0,0,0,0,0,0,0,0,0,0,0,0
P00033=-0.123,0.612,-5.012,0.0000,0.0000,0.0000
///RCONF 0,0,0,0,0,0,0,0,0,0,0,0,0,0,0,0,0,0,0,0,0,0,0,0
P00034=-0.304,0.773,-2.693,0.0000,0.0000,0.0000
P00035=2.817,0.591,-1.622,0.0000,0.0000,0.0000
P00036=-1.108,-0.829,1.850,0.0000,0.0000,0.0000
P00037=0.023,0.937,-2.677,0.0000,0.0000,0.0000
P00038=0.158,-1.133,-1.952,0.0000,0.0000,0.0000
P00039=0.012,-3.081,-0.106,0.0000,0.0000,0.0000
P00040=-0.030,9.648,2.467,0.0000,0.0000,0.0000
P00041=0.192,3.924,0.305,0.0000,0.0000,0.0000
P00042=-0.217,1.941,0.413,0.0000,0.0000,0.0000
P00043=-0.044,-1.937,1.197,0.0000,0.0000,0.0000
P00044=0.687,-2.322,1.156,0.0000,0.0000,0.0000
P00045=-0.068,-0.810,1.603,0.0000,0.0000,0.0000
P00046=0.799,0.043,1.292,0.0000,0.0000,0.0000
///RCONF 0,1,0,0,0,0,0,0,0,0,0,0,0,0,0,0,0,0,0,0,0,0,0,0
P00047=-0.011,1.737,-0.646,0.0000,0.0000,0.0000
///RCONF 0,0,0,0,0,0,0,0,0,0,0,0,0,0,0,0,0,0,0,0,0,0,0,0
P00048=2.411,0.025,-0.606,0.0000,0.0000,0.0000
P00049=3.413,-3.572,-1.618,0.0000,0.0000,0.0000
P00050=4.296,-4.501,-0.826,0.0000,0.0000,0.0000
P00051=0.367,3.892,0.009,0.0000,0.0000,0.0000
P00052=0.088,2.832,-0.342,0.0000,0.0000,0.0000
P00053=0.134,6.594,0.107,0.0000,0.0000,0.0000
P00054=-0.103,6.509,-0.702,0.0000,0.0000,0.0000
P00055=-0.342,8.912,1.324,0.0000,0.0000,0.0000
P00061=1.575,-3.405,-0.752,0.0000,0.0000,0.0000
P00062=-0.135,-0.848,-1.706,0.0000,0.0000,0.0000
P00063=0.036,-0.654,-3.005,0.0000,0.0000,0.0000
P00069=2.004,-0.013,0.498,0.0000,0.0000,0.0000
P00071=2.716,0.070,1.352,0.0000,0.0000,0.0000
P00072=1.041,-0.003,-0.797,0.0000,0.0000,0.0000
P00073=-0.961,5.319,-6.157,0.0000,0.0000,0.0000
P00074=1.123,1.944,-5.914,0.0000,0.0000,0.0000
P00080=-3.893,-3.240,-0.208,0.0000,0.0000,0.0000
P00081=19.486,11.347,1.262,0.0000,0.0000,0.0000
P00095=-3.945,4.918,-0.177,0.0000,0.0000,0.0000
P00096=-0.633,5.398,-3.809,0.0000,0.0000,0.0000
P00097=0.069,0.776,0.128,0.0000,0.0000,0.0000
P00098=0.276,2.477,1.230,0.0000,0.0000,0.0000
//INST
///DATE 2025/04/04 12:58
///ATTR SC,RW
///GROUP1 RB1,BS1
///GROUP2 ST1
NOP
'X2_8A-21A(90,0)
MOVJ C00000 BC00000 VJ=100.00  +MOVJ EC00000 VJ=100.00
CALL JOB:CLEAN-R1_KM_3P
MOVJ C00001 BC00001 VJ=100.00  +MOVJ EC00001 VJ=100.00
MOVJ C00002 BC00002 VJ=100.00  +MOVJ EC00002 VJ=100.00
'Path S3463
SFTOF3D
MOVJ C00003 BC00003 VJ=100.00  +MOVJ EC00003 VJ=100.00
MOVL C00004 BC00004 V=666.7  +MOVJ EC00004 VJ=100.00
SMOVL C00005 BC00005 V=166.7  +MOVJ EC00005
SREFP 3 C00006 BC00006  +REFP EC00006
CALL JOB:SEARCH-R1-S13D
SET P095 P006
SFTON3D P095
SMOVL C00007 BC00007 V=166.7  +MOVJ EC00007
SMOVL C00008 BC00008 V=166.7  +MOVJ EC00008
SREFP 3 C00009 BC00009  +REFP EC00009
CALL JOB:SEARCH-R1-S13D
SET P095 P006
SFTON3D P095
SMOVL C00010 BC00010 V=166.7  +MOVJ EC00010
MOVL C00011 BC00011 V=1000.0  +MOVJ EC00011 VJ=100.00
'EndPath S3463
'Path S3464
SFTOF3D
MOVJ C00012 BC00012 VJ=100.00  +MOVJ EC00012 VJ=100.00
MOVL C00013 BC00013 V=666.7  +MOVJ EC00013 VJ=100.00
SMOVL C00014 BC00014 V=166.7  +MOVJ EC00014
SREFP 3 C00015 BC00015  +REFP EC00015
CALL JOB:SEARCH-R1-S13D
SET P096 P006
SFTON3D P096
SMOVL C00016 BC00016 V=166.7  +MOVJ EC00016
SREFP 3 C00017 BC00017  +REFP EC00017
CALL JOB:SEARCH-R1-S13D
SET P096 P006
SFTON3D P096
SMOVL C00018 BC00018 V=166.7  +MOVJ EC00018
MOVL C00019 BC00019 V=1000.0  +MOVJ EC00019 VJ=100.00
'EndPath S3464
'Path S3465
SFTOF3D
MOVJ C00020 BC00020 VJ=100.00  +MOVJ EC00020 VJ=100.00
MOVL C00021 BC00021 V=666.7  +MOVJ EC00021 VJ=100.00
MOVL C00022 BC00022 V=666.7  +MOVJ EC00022 VJ=100.00
SMOVL C00023 BC00023 V=166.7  +MOVJ EC00023
SREFP 3 C00024 BC00024  +REFP EC00024
CALL JOB:SEARCH-R1-S13D
SET P097 P006
SFTON3D P097
SMOVL C00025 BC00025 V=166.7  +MOVJ EC00025
SMOVL C00026 BC00026 V=166.7  +MOVJ EC00026
SREFP 3 C00027 BC00027  +REFP EC00027
CALL JOB:SEARCH-R1-S13D
SET P097 P006
SFTON3D P097
SMOVL C00028 BC00028 V=166.7  +MOVJ EC00028
SMOVL C00029 BC00029 V=166.7  +MOVJ EC00029
SREFP 3 C00030 BC00030  +REFP EC00030
CALL JOB:SEARCH-R1-S13D
SET P021 P006
SFTON3D P021
SMOVL C00031 BC00031 V=166.7  +MOVJ EC00031
SMOVL C00032 BC00032 V=166.7  +MOVJ EC00032
SREFP 3 C00033 BC00033  +REFP EC00033
CALL JOB:SEARCH-R1-S13D
SET P021 P006
SFTON3D P021
SMOVL C00034 BC00034 V=166.7  +MOVJ EC00034
MOVL C00035 BC00035 V=1000.0  +MOVJ EC00035 VJ=100.00
'EndPath S3465
'Path S3464
SFTOF3D
MOVJ C00036 BC00036 VJ=100.00  +MOVJ EC00036 VJ=100.00
MOVL C00037 BC00037 V=666.7  +MOVJ EC00037 VJ=100.00
SMOVL C00038 BC00038 V=166.7  +MOVJ EC00038
SREFP 3 C00039 BC00039  +REFP EC00039
CALL JOB:SEARCH-R1-S13D
SET P022 P006
SFTON3D P022
SMOVL C00040 BC00040 V=166.7  +MOVJ EC00040
SREFP 3 C00041 BC00041  +REFP EC00041
CALL JOB:SEARCH-R1-S13D
SET P022 P006
SFTON3D P022
SMOVL C00042 BC00042 V=166.7  +MOVJ EC00042
MOVL C00043 BC00043 V=1000.0  +MOVJ EC00043 VJ=100.00
'EndPath S3464
MOVJ C00044 BC00044 VJ=100.00  +MOVJ EC00044 VJ=100.00
'Path S3465
SFTOF3D
MOVJ C00045 BC00045 VJ=100.00  +MOVJ EC00045 VJ=100.00
MOVL C00046 BC00046 V=666.7  +MOVJ EC00046 VJ=100.00
SMOVL C00047 BC00047 V=166.7  +MOVJ EC00047
SREFP 3 C00048 BC00048  +REFP EC00048
CALL JOB:SEARCH-R1-S13D
SET P050 P006
SFTON3D P050
SMOVL C00049 BC00049 V=166.7  +MOVJ EC00049
SREFP 3 C00050 BC00050  +REFP EC00050
CALL JOB:SEARCH-R1-S13D
SET P050 P006
SFTON3D P050
SMOVL C00051 BC00051 V=166.7  +MOVJ EC00051
SMOVL C00052 BC00052 V=166.7  +MOVJ EC00052
SREFP 3 C00053 BC00053  +REFP EC00053
CALL JOB:SEARCH-R1-S13D
SET P050 P006
SFTON3D P050
SMOVL C00054 BC00054 V=166.7  +MOVJ EC00054
MOVL C00055 BC00055 V=1000.0  +MOVJ EC00055 VJ=100.00
'EndPath S3465
'Path S3466
SFTOF3D
MOVJ C00056 BC00056 VJ=100.00  +MOVJ EC00056 VJ=100.00
MOVL C00057 BC00057 V=666.7  +MOVJ EC00057 VJ=100.00
SMOVL C00058 BC00058 V=166.7  +MOVJ EC00058
SREFP 3 C00059 BC00059  +REFP EC00059
CALL JOB:SEARCH-R1-S13D
SET P051 P006
SFTON3D P051
SMOVL C00060 BC00060 V=166.7  +MOVJ EC00060
SREFP 3 C00061 BC00061  +REFP EC00061
CALL JOB:SEARCH-R1-S13D
SET P051 P006
SFTON3D P051
SMOVL C00062 BC00062 V=166.7  +MOVJ EC00062
SMOVL C00063 BC00063 V=250.0  +MOVJ EC00063
SREFP 3 C00064 BC00064  +REFP EC00064
CALL JOB:SEARCH-R1-S13D
SET P051 P006
SFTON3D P051
SMOVL C00065 BC00065 V=166.7  +MOVJ EC00065
MOVL C00066 BC00066 V=1000.0  +MOVJ EC00066 VJ=100.00
'EndPath S3466
MOVJ C00067 BC00067 VJ=100.00  +MOVJ EC00067 VJ=100.00
MOVJ C00068 BC00068 VJ=100.00  +MOVJ EC00068 VJ=100.00
'Path S3467
SFTOF3D
MOVJ C00069 BC00069 VJ=100.00  +MOVJ EC00069 VJ=100.00
MOVL C00070 BC00070 V=666.7  +MOVJ EC00070 VJ=100.00
SMOVL C00071 BC00071 V=166.7  +MOVJ EC00071
SREFP 3 C00072 BC00072  +REFP EC00072
CALL JOB:SEARCH-R1-S13D
SET P054 P006
SFTON3D P054
SMOVL C00073 BC00073 V=250.0  +MOVJ EC00073
SMOVL C00074 BC00074 V=166.7  +MOVJ EC00074
SREFP 3 C00075 BC00075  +REFP EC00075
CALL JOB:SEARCH-R1-S13D
SET P054 P006
SFTON3D P054
SMOVL C00076 BC00076 V=166.7  +MOVJ EC00076
SMOVL C00077 BC00077 V=800.0  +MOVJ EC00077
SMOVL C00078 BC00078 V=166.7  +MOVJ EC00078
SREFP 3 C00079 BC00079  +REFP EC00079
CALL JOB:SEARCH-R1-S13D
SET P054 P006
SFTON3D P054
SMOVL C00080 BC00080 V=166.7  +MOVJ EC00080
MOVL C00081 BC00081 V=1000.0  +MOVJ EC00081 VJ=100.00
'EndPath S3467
'Path S3475
SFTOF3D
MOVJ C00082 BC00082 VJ=100.00  +MOVJ EC00082 VJ=100.00
MOVL C00083 BC00083 V=666.7  +MOVJ EC00083 VJ=100.00
SMOVL C00084 BC00084 V=166.7  +MOVJ EC00084
SREFP 3 C00085 BC00085  +REFP EC00085
CALL JOB:SEARCH-R1-S13D
SET P034 P006
SFTON3D P034
SMOVL C00086 BC00086 V=166.7  +MOVJ EC00086
SMOVL C00087 BC00087 V=333.3  +MOVJ EC00087
SMOVL C00088 BC00088 V=166.7  +MOVJ EC00088
SREFP 3 C00089 BC00089  +REFP EC00089
CALL JOB:SEARCH-R1-S13D
SET P034 P006
SFTON3D P034
SMOVL C00090 BC00090 V=166.7  +MOVJ EC00090
SMOVL C00091 BC00091 V=166.7  +MOVJ EC00091
SREFP 3 C00092 BC00092  +REFP EC00092
CALL JOB:SEARCH-R1-S13D
SET P034 P006
SFTON3D P034
SMOVL C00093 BC00093 V=166.7  +MOVJ EC00093
MOVL C00094 BC00094 V=1000.0  +MOVJ EC00094 VJ=100.00
'EndPath S3475
'Path S3464
SFTOF3D
MOVJ C00095 BC00095 VJ=100.00  +MOVJ EC00095 VJ=100.00
MOVL C00096 BC00096 V=666.7  +MOVJ EC00096 VJ=100.00
SMOVL C00097 BC00097 V=166.7  +MOVJ EC00097
SREFP 3 C00098 BC00098  +REFP EC00098
CALL JOB:SEARCH-R1-S13D
SET P023 P006
SFTON3D P023
SMOVL C00099 BC00099 V=166.7  +MOVJ EC00099
SMOVL C00100 BC00100 V=500.0  +MOVJ EC00100
SMOVL C00101 BC00101 V=166.7  +MOVJ EC00101
SREFP 3 C00102 BC00102  +REFP EC00102
CALL JOB:SEARCH-R1-S13D
SET P023 P006
SFTON3D P023
SMOVL C00103 BC00103 V=166.7  +MOVJ EC00103
SMOVL C00104 BC00104 V=166.7  +MOVJ EC00104
SREFP 3 C00105 BC00105  +REFP EC00105
CALL JOB:SEARCH-R1-S13D
SET P023 P006
SFTON3D P023
SMOVL C00106 BC00106 V=166.7  +MOVJ EC00106
MOVL C00107 BC00107 V=1000.0  +MOVJ EC00107 VJ=100.00
MOVJ C00108 BC00108 VJ=80.00  +MOVJ EC00108 VJ=80.00
MOVJ C00109 BC00109 VJ=80.00  +MOVJ EC00109 VJ=80.00
SFTOF3D
MOVJ C00110 BC00110 VJ=80.00  +MOVJ EC00110 VJ=80.00
SMOVL C00111 BC00111 V=166.7  +MOVJ EC00111
SREFP 3 C00112 BC00112  +REFP EC00112
CALL JOB:SEARCH-R1-S13D
SET P061 P006
SFTON3D P061
SMOVL C00113 BC00113 V=166.7  +MOVJ EC00113
SREFP 3 C00114 BC00114  +REFP EC00114
CALL JOB:SEARCH-R1-S13D
SET P061 P006
SFTON3D P061
SMOVL C00115 BC00115 V=166.7  +MOVJ EC00115
SFTOF3D
SMOVL C00116 BC00116 V=500.0  +MOVJ EC00116
SMOVL C00117 BC00117 V=166.7  +MOVJ EC00117
SREFP 3 C00118 BC00118  +REFP EC00118
CALL JOB:SEARCH-R1-S13D
SET P062 P006
SFTON3D P062
SMOVL C00119 BC00119 V=166.7  +MOVJ EC00119
SREFP 3 C00120 BC00120  +REFP EC00120
CALL JOB:SEARCH-R1-S13D
SET P062 P006
SFTON3D P062
SMOVL C00121 BC00121 V=166.7  +MOVJ EC00121
SFTOF3D
SMOVL C00122 BC00122 V=500.0  +MOVJ EC00122
SMOVL C00123 BC00123 V=166.7  +MOVJ EC00123
SREFP 3 C00124 BC00124  +REFP EC00124
CALL JOB:SEARCH-R1-S13D
SET P063 P006
SFTON3D P063
SMOVL C00125 BC00125 V=166.7  +MOVJ EC00125
SREFP 3 C00126 BC00126  +REFP EC00126
CALL JOB:SEARCH-R1-S13D
SET P063 P006
SFTON3D P063
SMOVL C00127 BC00127 V=166.7  +MOVJ EC00127
SFTOF3D
SMOVL C00128 BC00128 V=500.0  +MOVJ EC00128
MOVJ C00129 BC00129 VJ=80.00  +MOVJ EC00129 VJ=80.00
MOVJ C00130 BC00130 VJ=80.00  +MOVJ EC00130 VJ=80.00
'EndPath S3464
MOVJ C00131 BC00131 VJ=100.00  +MOVJ EC00131 VJ=100.00
'Path S3465
SFTOF3D
MOVJ C00132 BC00132 VJ=100.00  +MOVJ EC00132 VJ=100.00
MOVL C00133 BC00133 V=666.7  +MOVJ EC00133 VJ=100.00
SMOVL C00134 BC00134 V=166.7  +MOVJ EC00134
SREFP 3 C00135 BC00135  +REFP EC00135
CALL JOB:SEARCH-R1-S13D
SET P024 P006
SFTON3D P024
SMOVL C00136 BC00136 V=166.7  +MOVJ EC00136
SREFP 3 C00137 BC00137  +REFP EC00137
CALL JOB:SEARCH-R1-S13D
SET P024 P006
SFTON3D P024
SMOVL C00138 BC00138 V=166.7  +MOVJ EC00138
SMOVL C00139 BC00139 V=166.7  +MOVJ EC00139
SREFP 3 C00140 BC00140  +REFP EC00140
CALL JOB:SEARCH-R1-S13D
SET P024 P006
SFTON3D P024
SMOVL C00141 BC00141 V=166.7  +MOVJ EC00141
MOVL C00142 BC00142 V=1000.0  +MOVJ EC00142 VJ=100.00
'EndPath S3465
'Path S3476
MOVL C00143 BC00143 V=666.7  +MOVJ EC00143 VJ=100.00
SMOVL C00144 BC00144 V=166.7  +MOVJ EC00144
SREFP 3 C00145 BC00145  +REFP EC00145
CALL JOB:SEARCH-R1-S13D
SET P036 P006
SFTON3D P036
SMOVL C00146 BC00146 V=166.7  +MOVJ EC00146
SREFP 3 C00147 BC00147  +REFP EC00147
CALL JOB:SEARCH-R1-S13D
SET P036 P006
SFTON3D P036
SMOVL C00148 BC00148 V=166.7  +MOVJ EC00148
MOVL C00149 BC00149 V=666.7  +MOVJ EC00149 VJ=100.00
SFTOF3D
MOVJ C00150 BC00150 VJ=100.00  +MOVJ EC00150 VJ=100.00
MOVL C00151 BC00151 V=666.7  +MOVJ EC00151 VJ=100.00
SMOVL C00152 BC00152 V=166.7  +MOVJ EC00152
SREFP 3 C00153 BC00153  +REFP EC00153
CALL JOB:SEARCH-R1-S13D
SET P035 P006
SFTON3D P035
SMOVL C00154 BC00154 V=166.7  +MOVJ EC00154
SREFP 3 C00155 BC00155  +REFP EC00155
CALL JOB:SEARCH-R1-S13D
SET P035 P006
SFTON3D P035
SMOVL C00156 BC00156 V=166.7  +MOVJ EC00156
SMOVL C00157 BC00157 V=333.3  +MOVJ EC00157
SMOVL C00158 BC00158 V=166.7  +MOVJ EC00158
SREFP 3 C00159 BC00159  +REFP EC00159
CALL JOB:SEARCH-R1-S13D
SET P035 P006
SFTON3D P035
SMOVL C00160 BC00160 V=166.7  +MOVJ EC00160
MOVL C00161 BC00161 V=1000.0  +MOVJ EC00161 VJ=100.00
'EndPath S3476
'Path S3470
SFTOF3D
MOVJ C00162 BC00162 VJ=100.00  +MOVJ EC00162 VJ=100.00
MOVL C00163 BC00163 V=666.7  +MOVJ EC00163 VJ=100.00
SMOVL C00164 BC00164 V=166.7  +MOVJ EC00164
SREFP 3 C00165 BC00165  +REFP EC00165
CALL JOB:SEARCH-R1-S13D
SET P029 P006
SFTON3D P029
SMOVL C00166 BC00166 V=166.7  +MOVJ EC00166
SREFP 3 C00167 BC00167  +REFP EC00167
CALL JOB:SEARCH-R1-S13D
SET P029 P006
SFTON3D P029
SMOVL C00168 BC00168 V=166.7  +MOVJ EC00168
MOVL C00169 BC00169 V=666.7  +MOVJ EC00169 VJ=100.00
SMOVL C00170 BC00170 V=166.7  +MOVJ EC00170
SREFP 3 C00171 BC00171  +REFP EC00171
CALL JOB:SEARCH-R1-S13D
SET P037 P006
SFTON3D P037
SMOVL C00172 BC00172 V=166.7  +MOVJ EC00172
SREFP 3 C00173 BC00173  +REFP EC00173
CALL JOB:SEARCH-R1-S13D
SET P037 P006
SFTON3D P037
SMOVL C00174 BC00174 V=166.7  +MOVJ EC00174
SREFP 3 C00175 BC00175  +REFP EC00175
CALL JOB:SEARCH-R1-S13D
SET P038 P006
SFTON3D P038
SMOVL C00176 BC00176 V=166.7  +MOVJ EC00176
SREFP 3 C00177 BC00177  +REFP EC00177
CALL JOB:SEARCH-R1-S13D
SET P038 P006
SFTON3D P038
SMOVL C00178 BC00178 V=166.7  +MOVJ EC00178
SMOVL C00179 BC00179 V=1000.0  +MOVJ EC00179
MOVL C00180 BC00180 V=666.7  +MOVJ EC00180 VJ=100.00
SMOVL C00181 BC00181 V=166.7  +MOVJ EC00181
SREFP 3 C00182 BC00182  +REFP EC00182
CALL JOB:SEARCH-R1-S13D
SET P039 P006
SFTON3D P039
SMOVL C00183 BC00183 V=166.7  +MOVJ EC00183
SREFP 3 C00184 BC00184  +REFP EC00184
CALL JOB:SEARCH-R1-S13D
SET P039 P006
SFTON3D P039
SMOVL C00185 BC00185 V=166.7  +MOVJ EC00185
MOVL C00186 BC00186 V=666.7  +MOVJ EC00186 VJ=100.00
SMOVL C00187 BC00187 V=166.7  +MOVJ EC00187
SREFP 3 C00188 BC00188  +REFP EC00188
CALL JOB:SEARCH-R1-S13D
SET P040 P006
SFTON3D P040
SMOVL C00189 BC00189 V=166.7  +MOVJ EC00189
SREFP 3 C00190 BC00190  +REFP EC00190
CALL JOB:SEARCH-R1-S13D
SET P040 P006
SFTON3D P040
SMOVL C00191 BC00191 V=166.7  +MOVJ EC00191
SREFP 3 C00192 BC00192  +REFP EC00192
CALL JOB:SEARCH-R1-S13D
SET P041 P006
SFTON3D P041
SMOVL C00193 BC00193 V=166.7  +MOVJ EC00193
SREFP 3 C00194 BC00194  +REFP EC00194
CALL JOB:SEARCH-R1-S13D
SET P041 P006
SFTON3D P041
